KUKA KRL program: MyProgram_138().src

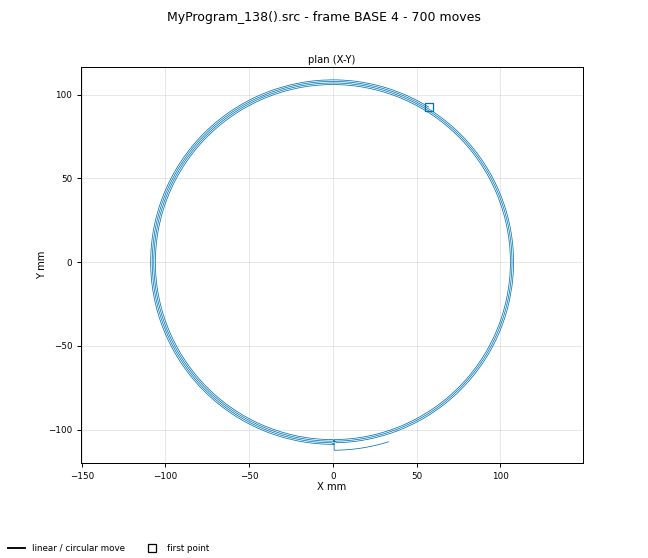
[picture p0: tool path of MyProgram_138().src in frame BASE 4, 700 of 700 moves have a stored position in this frame; points joined in program order, loops and branches not executed]
&ACCESS RVP
&REL 1
&PARAM TEMPLATE = C:\KRC\Roboter\Template\vorgabe
&PARAM EDITMASK = *
DEF MyProgram_138()
; ---- Setting reference (Base) ----
$BASE = BASE_DATA[4]

; --------------------------
; ---- Setting tool (TCP) ----
$TOOL = TOOL_DATA[3]
; --------------------------

$VEL.CP = VEL_APROX_PRINT
Startdeposition()
$VEL.CP = VEL_PRINT
LIN {X 57.2124,Y 92.5973,Z 111,A 54.04,B 24.9282,C -1.9571,E1 25.0833,E2 391.5977} C_DIS
LIN {X 54.554,Y 94.1872,Z 111,A 56.5809,B 24.9251,C -1.9983,E1 25.0769,E2 388.9668} C_DIS
LIN {X 49.9043,Y 96.7314,Z 111,A 58.528,B 24.9275,C -1.9661,E1 25.0723,E2 387.1015} C_DIS
LIN {X 44.6968,Y 99.2443,Z 111,A 61.4377,B 24.9277,C -1.9641,E1 25.065,E2 384.2041} C_DIS
LIN {X 41.4187,Y 100.6573,Z 111,A 63.4563,B 24.9271,C -1.9719,E1 25.0598,E2 382.1716} C_DIS
LIN {X 35.1577,Y 103.0113,Z 111,A 66.9301,B 24.9271,C -1.9732,E1 25.0507,E2 378.7021} C_DIS
LIN {X 31.9935,Y 104.0371,Z 111,A 68.7671,B 24.9266,C -1.9782,E1 25.0457,E2 376.8566} C_DIS
LIN {X 27.3515,Y 105.3527,Z 111,A 71.9417,B 24.9245,C -2.0064,E1 25.037,E2 373.6203} C_DIS
LIN {X 22.7022,Y 106.4523,Z 111,A 74.5175,B 24.9242,C -2.0101,E1 25.03,E2 371.0389} C_DIS
LIN {X 17.8344,Y 107.374,Z 111,A 76.2427,B 24.9269,C -1.9744,E1 25.0255,E2 369.4002} C_DIS
LIN {X 13.2214,Y 108.0405,Z 111,A 78.8231,B 24.9265,C -1.9802,E1 25.0183,E2 366.8082} C_DIS
LIN {X 10.1489,Y 108.3709,Z 111,A 80.4425,B 24.9265,C -1.9802,E1 25.0138,E2 365.1901} C_DIS
LIN {X 6.1973,Y 108.6686,Z 111,A 82.3574,B 24.927,C -1.9732,E1 25.0085,E2 363.2924} C_DIS
LIN {X 2.4816,Y 108.8177,Z 111,A 84.5086,B 24.9264,C -1.9809,E1 25.0024,E2 361.1235} C_DIS
LIN {X -0.9,Y 108.8415,Z 111,A 86.2853,B 24.9264,C -1.9804,E1 24.9975,E2 359.348} C_DIS
LIN {X -6.1677,Y 108.6702,Z 111,A 88.9687,B 24.9268,C -1.9758,E1 24.99,E2 356.675} C_DIS
LIN {X -8.9603,Y 108.4759,Z 111,A 90.5818,B 24.9264,C -1.9807,E1 24.9855,E2 355.0494} C_DIS
LIN {X -12.5967,Y 108.1136,Z 111,A 92.3889,B 24.9269,C -1.975,E1 24.9805,E2 353.2548} C_DIS
LIN {X -15.0336,Y 107.8021,Z 111,A 94.1095,B 24.9256,C -1.9914,E1 24.9757,E2 351.494} C_DIS
LIN {X -18.3991,Y 107.2796,Z 111,A 95.5312,B 24.9269,C -1.9751,E1 24.9718,E2 350.1095} C_DIS
LIN {X -25.1527,Y 105.9009,Z 111,A 99.3647,B 24.9265,C -1.9801,E1 24.9613,E2 346.2595} C_DIS
LIN {X -33.6723,Y 103.5057,Z 111,A 103.7876,B 24.9276,C -1.9656,E1 24.9496,E2 341.8638} C_DIS
LIN {X -37.933,Y 102.0233,Z 111,A 107.1546,B 24.9249,C -2.0019,E1 24.9405,E2 338.4036} C_DIS
LIN {X -43.1716,Y 99.9178,Z 111,A 109.1699,B 24.928,C -1.9597,E1 24.9355,E2 336.484} C_DIS
LIN {X -45.8586,Y 98.7129,Z 111,A 111.3295,B 24.9264,C -1.9813,E1 24.9299,E2 334.2676} C_DIS
LIN {X -49.6292,Y 96.872,Z 111,A 113.0255,B 24.9282,C -1.9575,E1 24.9258,E2 332.6237} C_DIS
LIN {X -53.729,Y 94.6613,Z 111,A 115.5042,B 24.9284,C -1.9543,E1 24.9198,E2 330.1455} C_DIS
LIN {X -56.0407,Y 93.3113,Z 111,A 117.2675,B 24.9276,C -1.9655,E1 24.9155,E2 328.3501} C_DIS
LIN {X -58.9868,Y 91.4759,Z 111,A 119.0332,B 24.928,C -1.9596,E1 24.9114,E2 326.5927} C_DIS
LIN {X -61.7031,Y 89.6661,Z 111,A 120.854,B 24.928,C -1.9602,E1 24.9072,E2 324.7644} C_DIS
LIN {X -64.732,Y 87.5059,Z 111,A 122.4158,B 24.9294,C -1.9407,E1 24.9037,E2 323.2435} C_DIS
LIN {X -66.7485,Y 85.9768,Z 111,A 124.0953,B 24.9286,C -1.9513,E1 24.9,E2 321.5326} C_DIS
LIN {X -69.373,Y 83.873,Z 111,A 126.0861,B 24.9283,C -1.9559,E1 24.8956,E2 319.5231} C_DIS
LIN {X -72.5974,Y 81.0977,Z 111,A 127.7779,B 24.9302,C -1.9296,E1 24.8922,E2 317.8873} C_DIS
LIN {X -74.913,Y 78.9651,Z 111,A 130.0033,B 24.9289,C -1.9476,E1 24.8876,E2 315.6099} C_DIS
LIN {X -77.9708,Y 75.9481,Z 111,A 132.276,B 24.9293,C -1.9425,E1 24.8832,E2 313.3397} C_DIS
LIN {X -80.856,Y 72.8675,Z 111,A 133.8967,B 24.9313,C -1.9138,E1 24.8803,E2 311.7802} C_DIS
LIN {X -83.2813,Y 70.0844,Z 111,A 136.3565,B 24.9303,C -1.9285,E1 24.8757,E2 309.2742} C_DIS
LIN {X -85.66,Y 67.1548,Z 111,A 138.0787,B 24.9314,C -1.9131,E1 24.8728,E2 307.5805} C_DIS
LIN {X -89.1664,Y 62.4237,Z 111,A 140.7257,B 24.9332,C -1.8874,E1 24.8685,E2 304.9819} C_DIS
LIN {X -92.2646,Y 57.745,Z 111,A 143.568,B 24.9341,C -1.8748,E1 24.8642,E2 302.1553} C_DIS
LIN {X -94.6562,Y 53.7379,Z 111,A 146.4084,B 24.9336,C -1.8821,E1 24.8601,E2 299.2828} C_DIS
LIN {X -96.2307,Y 50.8616,Z 111,A 147.9789,B 24.9344,C -1.8712,E1 24.8581,E2 297.73} C_DIS
LIN {X -98.007,Y 47.3488,Z 111,A 150.5224,B 24.9335,C -1.8828,E1 24.8549,E2 295.1451} C_DIS
LIN {X -99.9574,Y 43.0809,Z 111,A 152.8141,B 24.9346,C -1.8685,E1 24.8523,E2 292.875} C_DIS
LIN {X -101.0893,Y 40.3553,Z 111,A 154.9142,B 24.9334,C -1.8844,E1 24.8501,E2 290.7251} C_DIS
LIN {X -102.593,Y 36.3596,Z 111,A 156.5128,B 24.9356,C -1.8529,E1 24.8486,E2 289.1927} C_DIS
LIN {X -103.8004,Y 32.7566,Z 111,A 159.3428,B 24.9339,C -1.878,E1 24.8462,E2 286.2866} C_DIS
LIN {X -105.1746,Y 28.0297,Z 111,A 161.1618,B 24.9365,C -1.8405,E1 24.8449,E2 284.5465} C_DIS
LIN {X -105.9982,Y 24.732,Z 111,A 162.9892,B 24.9368,C -1.8362,E1 24.8437,E2 282.7186} C_DIS
LIN {X -106.7148,Y 21.4336,Z 111,A 164.5554,B 24.9377,C -1.8226,E1 24.8428,E2 281.1756} C_DIS
LIN {X -107.3259,Y 18.1224,Z 111,A 166.8034,B 24.9369,C -1.8348,E1 24.8417,E2 278.8852} C_DIS
LIN {X -107.9826,Y 13.6782,Z 111,A 168.8208,B 24.9383,C -1.8141,E1 24.8409,E2 276.9052} C_DIS
LIN {X -108.6273,Y 6.8942,Z 111,A 172.2213,B 24.9396,C -1.7953,E1 24.8401,E2 273.5289} C_DIS
LIN {X -108.8458,Y 0.346,Z 111,A 176.3293,B 24.9387,C -1.8089,E1 24.8398,E2 269.364} C_DIS
LIN {X -108.7341,Y -4.9176,Z 111,A 179.5942,B 24.938,C -1.8187,E1 24.8402,E2 266.0559} C_DIS
LIN {X -108.3957,Y -9.8796,Z 111,A -178.6874,B 24.9409,C -1.7762,E1 24.8405,E2 264.4286} C_DIS
LIN {X -108.0842,Y -12.8483,Z 111,A -176.3822,B 24.9393,C -1.7989,E1 24.8413,E2 262.0553} C_DIS
LIN {X -107.5085,Y -17.0089,Z 111,A -175.2974,B 24.9426,C -1.7494,E1 24.8417,E2 261.0822} C_DIS
LIN {X -106.7448,Y -21.2874,Z 111,A -172.4521,B 24.9417,C -1.763,E1 24.8432,E2 258.1875} C_DIS
LIN {X -106.0513,Y -24.5023,Z 111,A -170.6918,B 24.942,C -1.7588,E1 24.8442,E2 256.4271} C_DIS
LIN {X -105.1166,Y -28.2445,Z 111,A -168.6801,B 24.9425,C -1.7518,E1 24.8456,E2 254.4202} C_DIS
LIN {X -104.1481,Y -31.6353,Z 111,A -166.8566,B 24.9429,C -1.7449,E1 24.8471,E2 252.6026} C_DIS
LIN {X -103.1613,Y -34.7129,Z 111,A -165.0914,B 24.9431,C -1.7422,E1 24.8486,E2 250.8337} C_DIS
LIN {X -101.8747,Y -38.3253,Z 111,A -163.07,B 24.9435,C -1.7363,E1 24.8505,E2 248.815} C_DIS
LIN {X -99.6824,Y -43.7115,Z 111,A -159.3421,B 24.9424,C -1.753,E1 24.8547,E2 245.0267} C_DIS
LIN {X -97.851,Y -47.6734,Z 111,A -157.5507,B 24.9441,C -1.727,E1 24.8568,E2 243.2875} C_DIS
LIN {X -96.043,Y -51.2181,Z 111,A -155.4476,B 24.9445,C -1.7216,E1 24.8595,E2 241.1863} C_DIS
LIN {X -94.3257,Y -54.313,Z 111,A -153.7803,B 24.9453,C -1.709,E1 24.8617,E2 239.54} C_DIS
LIN {X -92.4096,Y -57.5128,Z 111,A -151.6872,B 24.9453,C -1.7088,E1 24.8648,E2 237.4368} C_DIS
LIN {X -90.4268,Y -60.584,Z 111,A -149.6454,B 24.9453,C -1.7083,E1 24.868,E2 235.3858} C_DIS
LIN {X -88.0816,Y -63.9457,Z 111,A -147.5847,B 24.9459,C -1.6992,E1 24.8713,E2 233.3369} C_DIS
LIN {X -85.695,Y -67.1106,Z 111,A -145.4349,B 24.9461,C -1.6965,E1 24.8749,E2 231.1831} C_DIS
LIN {X -83.4977,Y -69.8247,Z 111,A -143.7557,B 24.9467,C -1.6861,E1 24.8779,E2 229.5211} C_DIS
LIN {X -79.5983,Y -74.2398,Z 111,A -140.4764,B 24.9467,C -1.6859,E1 24.884,E2 226.2275} C_DIS
LIN {X -77.1504,Y -76.7802,Z 111,A -138.7372,B 24.9473,C -1.6773,E1 24.8874,E2 224.5013} C_DIS
LIN {X -74.6706,Y -79.1931,Z 111,A -136.8281,B 24.9473,C -1.677,E1 24.8913,E2 222.5852} C_DIS
LIN {X -71.8231,Y -81.7849,Z 111,A -134.7808,B 24.9475,C -1.6737,E1 24.8955,E2 220.5374} C_DIS
LIN {X -69.7427,Y -83.5658,Z 111,A -132.6222,B 24.9459,C -1.6994,E1 24.9003,E2 218.3096} C_DIS
LIN {X -65.9899,Y -86.5614,Z 111,A -130.9059,B 24.9482,C -1.6626,E1 24.9039,E2 216.6744} C_DIS
LIN {X -63.1094,Y -88.6818,Z 111,A -129.01,B 24.9484,C -1.6599,E1 24.9082,E2 214.7784} C_DIS
LIN {X -59.8794,Y -90.8938,Z 111,A -126.8554,B 24.9484,C -1.6603,E1 24.9132,E2 212.6157} C_DIS
LIN {X -57.6029,Y -92.3533,Z 111,A -124.5906,B 24.9464,C -1.6918,E1 24.9188,E2 210.2688} C_DIS
LIN {X -53.1291,Y -94.9975,Z 111,A -122.724,B 24.9488,C -1.653,E1 24.9231,E2 208.4889} C_DIS
LIN {X -50.1806,Y -96.5888,Z 111,A -120.7064,B 24.9483,C -1.6608,E1 24.9281,E2 206.4471} C_DIS
LIN {X -46.4955,Y -98.4164,Z 111,A -118.5097,B 24.9483,C -1.6595,E1 24.9337,E2 204.2479} C_DIS
LIN {X -42.476,Y -100.2151,Z 111,A -115.6875,B 24.9473,C -1.6775,E1 24.9411,E2 201.3763} C_DIS
LIN {X -37.9906,Y -102.0015,Z 111,A -113.8181,B 24.9491,C -1.6478,E1 24.9458,E2 199.5738} C_DIS
LIN {X -34.7676,Y -103.1428,Z 111,A -112.0211,B 24.9492,C -1.6462,E1 24.9505,E2 197.7772} C_DIS
LIN {X -31.6974,Y -104.1289,Z 111,A -110.4301,B 24.9496,C -1.6406,E1 24.9547,E2 196.1967} C_DIS
LIN {X -27.4497,Y -105.3275,Z 111,A -108.0258,B 24.9495,C -1.6424,E1 24.9612,E2 193.7843} C_DIS
LIN {X -20.9541,Y -106.8096,Z 111,A -104.6866,B 24.95,C -1.6338,E1 24.9703,E2 190.4613} C_DIS
LIN {X -17.1155,Y -107.492,Z 111,A -102.4094,B 24.9495,C -1.6424,E1 24.9766,E2 188.1616} C_DIS
LIN {X -13.3228,Y -108.0286,Z 111,A -100.3774,B 24.9495,C -1.6426,E1 24.9822,E2 186.1274} C_DIS
LIN {X -9.7573,Y -108.407,Z 111,A -98.512,B 24.9495,C -1.6416,E1 24.9874,E2 184.2635} C_DIS
LIN {X -6.19,Y -108.669,Z 111,A -96.7152,B 24.9497,C -1.6381,E1 24.9924,E2 182.4744} C_DIS
LIN {X -2.5967,Y -108.8156,Z 111,A -94.7193,B 24.9494,C -1.6426,E1 24.998,E2 180.4676} C_DIS
LIN {X 0.7454,Y -108.8411,Z 111,A -93.1023,B 24.9498,C -1.6371,E1 25.0025,E2 178.8636} C_DIS
Enddeposition()
LIN {X 0.7454,Y -108.8411,Z 111,A -93.1023,B 24.9498,C -1.6371,E1 25.0025,E2 178.8636} C_DIS
Startdeposition()
$VEL.CP = VEL_PRINT
LIN {X -0.738,Y -107.9051,Z 111,A -94.6413,B 24.9507,C -1.6223,E1 24.9981,E2 180.4376} C_DIS
LIN {X -4.3276,Y -107.8213,Z 111,A -96.6193,B 24.9509,C -1.6192,E1 24.9925,E2 182.4233} C_DIS
LIN {X -7.8193,Y -107.6253,Z 111,A -98.4701,B 24.9509,C -1.6193,E1 24.9874,E2 184.2744} C_DIS
LIN {X -11.2609,Y -107.3185,Z 111,A -100.1986,B 24.9506,C -1.6238,E1 24.9826,E2 185.9932} C_DIS
LIN {X -14.047,Y -106.9896,Z 111,A -101.7202,B 24.9506,C -1.6228,E1 24.9784,E2 187.5184} C_DIS
LIN {X -18.1316,Y -106.374,Z 111,A -103.9669,B 24.9508,C -1.6212,E1 24.9722,E2 189.7707} C_DIS
LIN {X -23.6715,Y -105.2811,Z 111,A -106.8512,B 24.9504,C -1.627,E1 24.9643,E2 192.6447} C_DIS
LIN {X -29.1742,Y -103.8893,Z 111,A -109.9817,B 24.9506,C -1.6242,E1 24.9558,E2 195.7865} C_DIS
LIN {X -32.344,Y -102.947,Z 111,A -111.6626,B 24.9503,C -1.6284,E1 24.9513,E2 197.4602} C_DIS
LIN {X -35.3965,Y -101.9376,Z 111,A -113.4529,B 24.9504,C -1.6265,E1 24.9466,E2 199.2583} C_DIS
LIN {X -38.4461,Y -100.8267,Z 111,A -115.561,B 24.9512,C -1.613,E1 24.941,E2 201.4029} C_DIS
LIN {X -41.5207,Y -99.6005,Z 111,A -117.0017,B 24.9504,C -1.6272,E1 24.9373,E2 202.8132} C_DIS
LIN {X -45.2004,Y -97.9853,Z 111,A -119.114,B 24.9502,C -1.6304,E1 24.932,E2 204.9229} C_DIS
LIN {X -48.3907,Y -96.4494,Z 111,A -120.8123,B 24.9496,C -1.6398,E1 24.9278,E2 206.6033} C_DIS
LIN {X -50.5517,Y -95.3346,Z 111,A -122.1778,B 24.9496,C -1.6386,E1 24.9244,E2 207.9754} C_DIS
LIN {X -53.5282,Y -93.6956,Z 111,A -124.5217,B 24.9508,C -1.6202,E1 24.9185,E2 210.3699} C_DIS
LIN {X -56.6609,Y -91.8366,Z 111,A -125.887,B 24.9493,C -1.645,E1 24.9154,E2 211.6805} C_DIS
LIN {X -59.0124,Y -90.3427,Z 111,A -127.9307,B 24.9505,C -1.6256,E1 24.9105,E2 213.7769} C_DIS
LIN {X -61.8911,Y -88.3951,Z 111,A -129.5546,B 24.9498,C -1.6372,E1 24.9068,E2 215.3789} C_DIS
LIN {X -65.3162,Y -85.8967,Z 111,A -132.1133,B 24.9503,C -1.6294,E1 24.9011,E2 217.9652} C_DIS
LIN {X -68.1893,Y -83.6313,Z 111,A -133.7977,B 24.9494,C -1.6429,E1 24.8975,E2 219.6239} C_DIS
LIN {X -70.9889,Y -81.2689,Z 111,A -135.4897,B 24.9486,C -1.6563,E1 24.8939,E2 221.2906} C_DIS
LIN {X -73.785,Y -78.7392,Z 111,A -137.4949,B 24.9483,C -1.6602,E1 24.8898,E2 223.2946} C_DIS
LIN {X -76.3182,Y -76.289,Z 111,A -139.5037,B 24.9484,C -1.6589,E1 24.8858,E2 225.3149} C_DIS
LIN {X -78.7402,Y -73.784,Z 111,A -141.8483,B 24.9493,C -1.6444,E1 24.8812,E2 227.7043} C_DIS
LIN {X -81.5145,Y -70.7077,Z 111,A -143.5604,B 24.9479,C -1.6677,E1 24.8782,E2 229.3686} C_DIS
LIN {X -83.3934,Y -68.4835,Z 111,A -145.1511,B 24.9478,C -1.6696,E1 24.8753,E2 230.962} C_DIS
LIN {X -85.797,Y -65.4463,Z 111,A -147.1473,B 24.9473,C -1.6769,E1 24.8719,E2 232.9504} C_DIS
LIN {X -87.9068,Y -62.5816,Z 111,A -148.9056,B 24.9467,C -1.6865,E1 24.8691,E2 234.6943} C_DIS
LIN {X -90.3725,Y -58.9672,Z 111,A -151.3572,B 24.9467,C -1.6877,E1 24.8652,E2 237.1555} C_DIS
LIN {X -92.9979,Y -54.7311,Z 111,A -153.8722,B 24.9459,C -1.6996,E1 24.8616,E2 239.655} C_DIS
LIN {X -94.4729,Y -52.1461,Z 111,A -155.6836,B 24.9461,C -1.6952,E1 24.8591,E2 241.4862} C_DIS
LIN {X -96.2263,Y -48.833,Z 111,A -157.6728,B 24.9458,C -1.7008,E1 24.8565,E2 243.4728} C_DIS
LIN {X -98.6358,Y -43.7656,Z 111,A -160.669,B 24.9453,C -1.7086,E1 24.853,E2 246.4666} C_DIS
LIN {X -100.5834,Y -39.0793,Z 111,A -163.1815,B 24.9443,C -1.7233,E1 24.8504,E2 248.9583} C_DIS
LIN {X -101.5717,Y -36.4359,Z 111,A -164.901,B 24.9446,C -1.7195,E1 24.8487,E2 250.6964} C_DIS
LIN {X -102.7174,Y -33.064,Z 111,A -166.6168,B 24.9438,C -1.7317,E1 24.8472,E2 252.393} C_DIS
LIN {X -103.7009,Y -29.839,Z 111,A -168.5725,B 24.9438,C -1.731,E1 24.8457,E2 254.3616} C_DIS
LIN {X -104.6185,Y -26.4426,Z 111,A -170.4521,B 24.9435,C -1.7363,E1 24.8444,E2 256.2395} C_DIS
LIN {X -105.5182,Y -22.5863,Z 111,A -172.3655,B 24.9426,C -1.7498,E1 24.8432,E2 258.132} C_DIS
LIN {X -106.0381,Y -20.0036,Z 111,A -174.1059,B 24.9431,C -1.7417,E1 24.8423,E2 259.9021} C_DIS
LIN {X -106.6664,Y -16.3207,Z 111,A -176.597,B 24.9439,C -1.7295,E1 24.8412,E2 262.437} C_DIS
LIN {X -107.2643,Y -11.7781,Z 111,A -178.288,B 24.9417,C -1.7642,E1 24.8407,E2 264.0554} C_DIS
LIN {X -107.75,Y -5.8312,Z 111,A 177.9183,B 24.9425,C -1.7517,E1 24.8399,E2 267.9018} C_DIS
LIN {X -107.89,Y -1.952,Z 111,A 176.4307,B 24.9407,C -1.7792,E1 24.8399,E2 269.3328} C_DIS
LIN {X -107.9017,Y 1.2877,Z 111,A 173.8525,B 24.9424,C -1.7536,E1 24.8399,E2 271.9876} C_DIS
LIN {X -107.7322,Y 6.154,Z 111,A 172.5435,B 24.9387,C -1.8084,E1 24.84,E2 273.1736} C_DIS
LIN {X -107.2342,Y 12.0474,Z 111,A 168.9032,B 24.9393,C -1.8002,E1 24.8409,E2 276.8555} C_DIS
LIN {X -106.4571,Y 17.6345,Z 111,A 165.8379,B 24.9388,C -1.8073,E1 24.8422,E2 279.922} C_DIS
LIN {X -105.8443,Y 21.0099,Z 111,A 164.0175,B 24.9384,C -1.8132,E1 24.8431,E2 281.7393} C_DIS
LIN {X -105.1387,Y 24.2879,Z 111,A 162.2901,B 24.9379,C -1.8208,E1 24.8442,E2 283.4585} C_DIS
LIN {X -104.3811,Y 27.3664,Z 111,A 160.6393,B 24.9374,C -1.8274,E1 24.8453,E2 285.1033} C_DIS
LIN {X -102.9089,Y 32.4669,Z 111,A 157.825,B 24.9368,C -1.8364,E1 24.8475,E2 287.9123} C_DIS
LIN {X -102.0759,Y 34.9982,Z 111,A 155.8643,B 24.9378,C -1.8209,E1 24.8493,E2 289.9212} C_DIS
LIN {X -100.9575,Y 38.1006,Z 111,A 154.5126,B 24.9365,C -1.8409,E1 24.8506,E2 291.2327} C_DIS
LIN {X -99.5516,Y 41.6369,Z 111,A 152.4306,B 24.9362,C -1.8449,E1 24.8528,E2 293.3169} C_DIS
LIN {X -98.0253,Y 45.1144,Z 111,A 150.432,B 24.9357,C -1.8517,E1 24.8551,E2 295.3103} C_DIS
LIN {X -95.5364,Y 50.1685,Z 111,A 147.6057,B 24.9347,C -1.8666,E1 24.8586,E2 298.1161} C_DIS
LIN {X -94.2246,Y 52.5907,Z 111,A 145.5303,B 24.936,C -1.8485,E1 24.8614,E2 300.2458} C_DIS
LIN {X -92.4493,Y 55.6543,Z 111,A 144.2671,B 24.934,C -1.8765,E1 24.8632,E2 301.4486} C_DIS
LIN {X -89.2122,Y 60.7067,Z 111,A 140.9249,B 24.9338,C -1.8797,E1 24.8683,E2 304.7999} C_DIS
LIN {X -85.9122,Y 65.2936,Z 111,A 137.8999,B 24.9332,C -1.887,E1 24.8732,E2 307.8223} C_DIS
LIN {X -83.5498,Y 68.2912,Z 111,A 135.9664,B 24.9326,C -1.8958,E1 24.8766,E2 309.7439} C_DIS
LIN {X -81.9069,Y 70.2527,Z 111,A 134.3441,B 24.9331,C -1.8896,E1 24.8795,E2 311.3885} C_DIS
LIN {X -79.3749,Y 73.1007,Z 111,A 132.1113,B 24.9333,C -1.8869,E1 24.8838,E2 313.6374} C_DIS
LIN {X -75.2518,Y 77.3401,Z 111,A 129.2233,B 24.932,C -1.9039,E1 24.8894,E2 316.4973} C_DIS
LIN {X -72.8042,Y 79.647,Z 111,A 127.2477,B 24.9322,C -1.9011,E1 24.8935,E2 318.4877} C_DIS
LIN {X -68.7496,Y 83.1723,Z 111,A 124.4574,B 24.9316,C -1.9098,E1 24.8994,E2 321.268} C_DIS
LIN {X -66.5195,Y 84.9674,Z 111,A 122.9827,B 24.9313,C -1.9148,E1 24.9026,E2 322.7363} C_DIS
LIN {X -63.6498,Y 87.1366,Z 111,A 120.3678,B 24.9329,C -1.8925,E1 24.9087,E2 325.4135} C_DIS
LIN {X -59.63,Y 89.9355,Z 111,A 118.7898,B 24.9297,C -1.9359,E1 24.9121,E2 326.8934} C_DIS
LIN {X -55.5862,Y 92.4906,Z 111,A 116.0946,B 24.9298,C -1.9348,E1 24.9185,E2 329.5999} C_DIS
LIN {X -53.447,Y 93.7422,Z 111,A 114.6018,B 24.9301,C -1.9304,E1 24.9221,E2 331.1075} C_DIS
LIN {X -48.8756,Y 96.2045,Z 111,A 111.429,B 24.9309,C -1.9193,E1 24.93,E2 334.3153} C_DIS
LIN {X -45.6455,Y 97.7781,Z 111,A 110.3349,B 24.9285,C -1.9533,E1 24.9326,E2 335.3315} C_DIS
LIN {X -38.3358,Y 100.8684,Z 111,A 105.8393,B 24.9288,C -1.9485,E1 24.9443,E2 339.8488} C_DIS
LIN {X -35.4539,Y 101.9174,Z 111,A 104.1595,B 24.9288,C -1.9485,E1 24.9487,E2 341.5317} C_DIS
LIN {X -30.921,Y 103.3828,Z 111,A 101.238,B 24.9297,C -1.9364,E1 24.9565,E2 344.4873} C_DIS
LIN {X -27.1414,Y 104.4389,Z 111,A 99.472,B 24.9287,C -1.9508,E1 24.9612,E2 346.2218} C_DIS
LIN {X -23.6603,Y 105.2837,Z 111,A 97.4588,B 24.9288,C -1.9482,E1 24.9667,E2 348.2438} C_DIS
LIN {X -19.8949,Y 106.059,Z 111,A 95.7104,B 24.9279,C -1.9613,E1 24.9714,E2 349.9631} C_DIS
LIN {X -14.7588,Y 106.8944,Z 111,A 92.8831,B 24.9279,C -1.9606,E1 24.9793,E2 352.7943} C_DIS
LIN {X -11.7408,Y 107.2682,Z 111,A 91.0802,B 24.9284,C -1.9542,E1 24.9843,E2 354.6138} C_DIS
LIN {X -8.2886,Y 107.5893,Z 111,A 89.3773,B 24.9279,C -1.9605,E1 24.989,E2 356.3025} C_DIS
LIN {X -4.4317,Y 107.8168,Z 111,A 87.1143,B 24.9285,C -1.9529,E1 24.9954,E2 358.5842} C_DIS
LIN {X -0.4353,Y 107.907,Z 111,A 85.1947,B 24.9279,C -1.9614,E1 25.0007,E2 360.4836} C_DIS
LIN {X 2.8838,Y 107.8693,Z 111,A 83.4912,B 24.9277,C -1.964,E1 25.0054,E2 362.1807} C_DIS
LIN {X 5.0706,Y 107.7893,Z 111,A 82.2144,B 24.928,C -1.9595,E1 25.009,E2 363.4679} C_DIS
LIN {X 8.5205,Y 107.5707,Z 111,A 80.419,B 24.9279,C -1.961,E1 25.014,E2 365.2587} C_DIS
LIN {X 11.9578,Y 107.2447,Z 111,A 78.184,B 24.9291,C -1.9447,E1 25.0203,E2 367.5308} C_DIS
LIN {X 16.6099,Y 106.6217,Z 111,A 75.8193,B 24.9288,C -1.9492,E1 25.0268,E2 369.8829} C_DIS
LIN {X 21.239,Y 105.7978,Z 111,A 73.4981,B 24.9283,C -1.9552,E1 25.0331,E2 372.1873} C_DIS
LIN {X 26.4088,Y 104.6272,Z 111,A 70.6942,B 24.9284,C -1.954,E1 25.0407,E2 374.9899} C_DIS
LIN {X 29.5337,Y 103.7875,Z 111,A 69.0654,B 24.9282,C -1.9565,E1 25.0451,E2 376.6102} C_DIS
LIN {X 32.6151,Y 102.8626,Z 111,A 67.2668,B 24.9286,C -1.9515,E1 25.0499,E2 378.4174} C_DIS
LIN {X 35.6864,Y 101.8359,Z 111,A 65.2529,B 24.9296,C -1.9381,E1 25.0553,E2 380.4591} C_DIS
LIN {X 38.7765,Y 100.7015,Z 111,A 63.9576,B 24.9284,C -1.9548,E1 25.0586,E2 381.712} C_DIS
LIN {X 42.2315,Y 99.301,Z 111,A 61.9507,B 24.9286,C -1.9516,E1 25.0638,E2 383.7218} C_DIS
LIN {X 46.2111,Y 97.5133,Z 111,A 59.738,B 24.9285,C -1.9531,E1 25.0694,E2 385.9253} C_DIS
LIN {X 48.5885,Y 96.3512,Z 111,A 58.086,B 24.9294,C -1.9412,E1 25.0735,E2 387.6012} C_DIS
LIN {X 53.6524,Y 93.6242,Z 111,A 55.1647,B 24.9293,C -1.9425,E1 25.0807,E2 390.511} C_DIS
LIN {X 56.3715,Y 92.0134,Z 111,A 53.3292,B 24.9299,C -1.9334,E1 25.0851,E2 392.3622} C_DIS
LIN {X 59.719,Y 89.8769,Z 111,A 51.2986,B 24.9299,C -1.9333,E1 25.0898,E2 394.3865} C_DIS
LIN {X 62.5438,Y 87.9338,Z 111,A 49.5654,B 24.9299,C -1.9338,E1 25.0938,E2 396.1123} C_DIS
LIN {X 65.2492,Y 85.9471,Z 111,A 47.6885,B 24.9304,C -1.9267,E1 25.098,E2 397.9994} C_DIS
LIN {X 69.1918,Y 82.8048,Z 111,A 45.2182,B 24.9301,C -1.9303,E1 25.1033,E2 400.4517} C_DIS
LIN {X 71.2958,Y 81.0009,Z 111,A 43.6626,B 24.9306,C -1.9239,E1 25.1066,E2 402.0165} C_DIS
LIN {X 73.9316,Y 78.6014,Z 111,A 41.802,B 24.9308,C -1.9214,E1 25.1104,E2 403.8754} C_DIS
LIN {X 76.3037,Y 76.3037,Z 111,A 39.9056,B 24.9315,C -1.9116,E1 25.1142,E2 405.787} C_DIS
LIN {X 78.694,Y 73.8332,Z 111,A 38.1583,B 24.9315,C -1.9109,E1 25.1176,E2 407.5284} C_DIS
LIN {X 81.3051,Y 70.9475,Z 111,A 36.1391,B 24.9317,C -1.9081,E1 25.1213,E2 409.545} C_DIS
LIN {X 83.7948,Y 67.989,Z 111,A 34.1002,B 24.932,C -1.9039,E1 25.125,E2 411.5846} C_DIS
LIN {X 86.0865,Y 65.0636,Z 111,A 32.1213,B 24.9324,C -1.8988,E1 25.1283,E2 413.566} C_DIS
LIN {X 88.6392,Y 61.5399,Z 111,A 29.886,B 24.9326,C -1.8962,E1 25.132,E2 415.7966} C_DIS
LIN {X 89.9593,Y 59.5939,Z 111,A 28.6161,B 24.9329,C -1.8921,E1 25.1339,E2 417.07} C_DIS
LIN {X 91.5625,Y 57.0998,Z 111,A 27.0118,B 24.9333,C -1.8866,E1 25.1363,E2 418.679} C_DIS
LIN {X 94.2304,Y 52.5803,Z 111,A 24.3994,B 24.9333,C -1.8866,E1 25.14,E2 421.2781} C_DIS
LIN {X 95.6737,Y 49.9077,Z 111,A 22.4295,B 24.9347,C -1.8668,E1 25.1426,E2 423.2843} C_DIS
LIN {X 98.0946,Y 44.9656,Z 111,A 19.7273,B 24.9346,C -1.8679,E1 25.1458,E2 425.9693} C_DIS
LIN {X 99.4483,Y 41.8818,Z 111,A 18.0013,B 24.9348,C -1.8655,E1 25.1477,E2 427.6917} C_DIS
LIN {X 100.7789,Y 38.5723,Z 111,A 15.9223,B 24.9357,C -1.8519,E1 25.1499,E2 429.7911} C_DIS
LIN {X 102.3459,Y 34.1973,Z 111,A 13.6726,B 24.9356,C -1.8539,E1 25.1519,E2 432.0234} C_DIS
LIN {X 103.5566,Y 30.3352,Z 111,A 10.857,B 24.938,C -1.8187,E1 25.1542,E2 434.9061} C_DIS
LIN {X 104.7105,Y 26.0776,Z 111,A 9.3373,B 24.9361,C -1.8469,E1 25.1553,E2 436.3504} C_DIS
LIN {X 105.6823,Y 21.802,Z 111,A 6.4794,B 24.9381,C -1.8167,E1 25.157,E2 439.2629} C_DIS
LIN {X 106.3218,Y 18.4435,Z 111,A 4.9475,B 24.9377,C -1.8232,E1 25.1577,E2 440.7706} C_DIS
LIN {X 106.9433,Y 14.4042,Z 111,A 3.0533,B 24.9373,C -1.8283,E1 25.1585,E2 442.6415} C_DIS
LIN {X 107.4354,Y 10.086,Z 111,A 0.6302,B 24.9382,C -1.8159,E1 25.1592,E2 445.0795} C_DIS
LIN {X 107.6816,Y 6.987,Z 111,A -1.1243,B 24.9389,C -1.8061,E1 25.1595,E2 446.8468} C_DIS
LIN {X 107.8569,Y 3.3087,Z 111,A -2.9103,B 24.9388,C -1.8072,E1 25.1597,E2 448.6196} C_DIS
LIN {X 107.9106,Y 0.0081,Z 111,A -4.8343,B 24.9397,C -1.794,E1 25.1597,E2 450.5633} C_DIS
LIN {X 107.842,Y -3.7943,Z 111,A -6.7379,B 24.9397,C -1.7925,E1 25.1597,E2 452.4591} C_DIS
LIN {X 107.6659,Y -7.2186,Z 111,A -8.5067,B 24.94,C -1.7888,E1 25.1593,E2 454.226} C_DIS
LIN {X 107.3472,Y -10.9862,Z 111,A -10.523,B 24.9405,C -1.7819,E1 25.1588,E2 456.2466} C_DIS
LIN {X 106.9455,Y -14.3875,Z 111,A -12.4959,B 24.9413,C -1.7693,E1 25.1581,E2 458.2377} C_DIS
LIN {X 105.4909,Y -22.7113,Z 111,A -16.5089,B 24.9409,C -1.7755,E1 25.1562,E2 462.2126} C_DIS
LIN {X 104.4457,Y -27.115,Z 111,A -19.0926,B 24.942,C -1.7599,E1 25.1544,E2 464.8182} C_DIS
LIN {X 103.8442,Y -29.3333,Z 111,A -20.3649,B 24.9424,C -1.7537,E1 25.1535,E2 466.0976} C_DIS
LIN {X 102.9047,Y -32.4804,Z 111,A -21.9992,B 24.9424,C -1.753,E1 25.1521,E2 467.7244} C_DIS
LIN {X 101.6954,Y -36.0867,Z 111,A -24.6286,B 24.9445,C -1.7202,E1 25.1497,E2 470.4164} C_DIS
LIN {X 100.3576,Y -39.6542,Z 111,A -26.1254,B 24.9435,C -1.7367,E1 25.1482,E2 471.8659} C_DIS
LIN {X 99.1494,Y -42.5887,Z 111,A -28.2204,B 24.945,C -1.7137,E1 25.1459,E2 474.0036} C_DIS
LIN {X 97.7747,Y -45.6529,Z 111,A -29.5044,B 24.9439,C -1.73,E1 25.1444,E2 475.2423} C_DIS
LIN {X 96.3857,Y -48.5209,Z 111,A -31.7511,B 24.9458,C -1.7008,E1 25.1416,E2 477.5458} C_DIS
LIN {X 94.6609,Y -51.8028,Z 111,A -33.1101,B 24.9445,C -1.7214,E1 25.1398,E2 478.8491} C_DIS
LIN {X 93.0872,Y -54.58,Z 111,A -34.8665,B 24.945,C -1.7138,E1 25.1374,E2 480.6144} C_DIS
LIN {X 91.0387,Y -57.9327,Z 111,A -37.6636,B 24.9473,C -1.6771,E1 25.1331,E2 483.4838} C_DIS
LIN {X 88.5039,Y -61.7345,Z 111,A -39.3636,B 24.9457,C -1.7016,E1 25.1305,E2 485.1177} C_DIS
LIN {X 84.8324,Y -66.6903,Z 111,A -42.3568,B 24.9455,C -1.7048,E1 25.1256,E2 488.089} C_DIS
LIN {X 80.6833,Y -71.6551,Z 111,A -46.0222,B 24.9467,C -1.6858,E1 25.1189,E2 491.7826} C_DIS
LIN {X 76.0688,Y -76.5357,Z 111,A -50.3761,B 24.9494,C -1.6433,E1 25.1102,E2 496.218} C_DIS
LIN {X 72.4483,Y -79.9732,Z 111,A -52.3282,B 24.9479,C -1.6667,E1 25.1064,E2 498.1069} C_DIS
LIN {X 67.3844,Y -84.2838,Z 111,A -55.9246,B 24.9486,C -1.656,E1 25.0986,E2 501.7149} C_DIS
LIN {X 64.2159,Y -86.7221,Z 111,A -57.7313,B 24.9481,C -1.6649,E1 25.0947,E2 503.4939} C_DIS
LIN {X 58.5115,Y -90.6671,Z 111,A -61.6113,B 24.949,C -1.6491,E1 25.0857,E2 507.3982} C_DIS
LIN {X 55.5622,Y -92.5052,Z 111,A -63.4501,B 24.9492,C -1.6459,E1 25.0813,E2 509.2389} C_DIS
LIN {X 52.5474,Y -94.2488,Z 111,A -65.8567,B 24.9509,C -1.6192,E1 25.0753,E2 511.7015} C_DIS
LIN {X 48.6146,Y -96.3378,Z 111,A -67.7018,B 24.9498,C -1.6369,E1 25.0708,E2 513.4995} C_DIS
LIN {X 42.3827,Y -99.2372,Z 111,A -71.0416,B 24.9493,C -1.6443,E1 25.0624,E2 516.8135} C_DIS
LIN {X 38.0322,Y -100.9834,Z 111,A -73.6631,B 24.9499,C -1.6352,E1 25.0555,E2 519.4506} C_DIS
LIN {X 34.7539,Y -102.1583,Z 111,A -75.5159,B 24.95,C -1.6327,E1 25.0506,E2 521.3058} C_DIS
LIN {X 31.6978,Y -103.1474,Z 111,A -77.5269,B 24.9509,C -1.618,E1 25.0452,E2 523.3479} C_DIS
LIN {X 24.2476,Y -105.1481,Z 111,A -81.3049,B 24.9504,C -1.6269,E1 25.0351,E2 527.0989} C_DIS
LIN {X 21.4218,Y -105.7603,Z 111,A -82.9754,B 24.9508,C -1.62,E1 25.0304,E2 528.7839} C_DIS
LIN {X 15.8967,Y -106.732,Z 111,A -85.7213,B 24.9504,C -1.6272,E1 25.0229,E2 531.5097} C_DIS
LIN {X 13.2093,Y -107.0981,Z 111,A -87.3335,B 24.9509,C -1.6192,E1 25.0184,E2 533.1395} C_DIS
LIN {X 9.947,Y -107.4482,Z 111,A -88.9821,B 24.9507,C -1.6221,E1 25.0139,E2 534.7802} C_DIS
LIN {X 6.2467,Y -107.7271,Z 111,A -91.015,B 24.9509,C -1.6187,E1 25.0082,E2 536.8204} C_DIS
LIN {X 2.5986,Y -107.8781,Z 111,A -92.9933,B 24.951,C -1.6164,E1 25.0026,E2 538.8037} C_DIS
LIN {X 2.5986,Y -107.8781,Z 111,A -92.9933,B 24.951,C -1.6164,E1 25.0026,E2 538.8037} C_DIS
Enddeposition()
LIN {X 0.7392,Y -106.965,Z 111,A -93.8206,B 24.9496,C -1.6392,E1 25.0005,E2 539.5768} C_DIS
Startdeposition()
$VEL.CP = VEL_PRINT
LIN {X 2.536,Y -106.9417,Z 111,A -92.2411,B 24.9481,C -1.6644,E1 25.0051,E2 537.9377} C_DIS
LIN {X 5.275,Y -106.842,Z 111,A -90.5193,B 24.9474,C -1.6754,E1 25.0099,E2 536.1905} C_DIS
LIN {X 9.3438,Y -106.5626,Z 111,A -88.4308,B 24.9476,C -1.6725,E1 25.0157,E2 534.1099} C_DIS
LIN {X 12.9354,Y -106.1865,Z 111,A -86.6457,B 24.9479,C -1.6675,E1 25.0206,E2 532.3379} C_DIS
LIN {X 16.3048,Y -105.7204,Z 111,A -84.0145,B 24.9457,C -1.7025,E1 25.0281,E2 529.6262} C_DIS
LIN {X 20.9634,Y -104.8976,Z 111,A -82.3489,B 24.9478,C -1.6684,E1 25.0325,E2 528.0435} C_DIS
LIN {X 23.9158,Y -104.2627,Z 111,A -79.5353,B 24.9445,C -1.7201,E1 25.0405,E2 525.1112} C_DIS
LIN {X 29.8014,Y -102.7364,Z 111,A -77.3853,B 24.9473,C -1.677,E1 25.046,E2 523.0669} C_DIS
LIN {X 32.3942,Y -101.9489,Z 111,A -75.7962,B 24.9468,C -1.6845,E1 25.0502,E2 521.463} C_DIS
LIN {X 36.0655,Y -100.7091,Z 111,A -73.9344,B 24.9472,C -1.6781,E1 25.0551,E2 519.6199} C_DIS
LIN {X 38.1305,Y -99.9439,Z 111,A -72.589,B 24.9467,C -1.6867,E1 25.0586,E2 518.257} C_DIS
LIN {X 41.3479,Y -98.6562,Z 111,A -70.5732,B 24.9461,C -1.6962,E1 25.0639,E2 516.2235} C_DIS
LIN {X 47.8215,Y -95.6863,Z 111,A -67.2559,B 24.947,C -1.6811,E1 25.0722,E2 512.9503} C_DIS
LIN {X 51.8391,Y -93.5707,Z 111,A -64.812,B 24.9467,C -1.6858,E1 25.0782,E2 510.5023} C_DIS
LIN {X 55.4481,Y -91.4777,Z 111,A -62.3238,B 24.9458,C -1.7007,E1 25.0843,E2 507.9865} C_DIS
LIN {X 58.247,Y -89.7231,Z 111,A -60.426,B 24.9452,C -1.7096,E1 25.0888,E2 506.0738} C_DIS
LIN {X 60.6308,Y -88.1296,Z 111,A -58.9709,B 24.9452,C -1.7093,E1 25.0921,E2 504.6245} C_DIS
LIN {X 63.5378,Y -86.0568,Z 111,A -57.1351,B 24.9452,C -1.71,E1 25.0962,E2 502.7934} C_DIS
LIN {X 66.2856,Y -83.9575,Z 111,A -55.1578,B 24.9446,C -1.7194,E1 25.1006,E2 500.8012} C_DIS
LIN {X 71.1383,Y -79.8878,Z 111,A -51.9962,B 24.9447,C -1.7172,E1 25.1073,E2 497.6571} C_DIS
LIN {X 75.5605,Y -75.7203,Z 111,A -48.8941,B 24.9447,C -1.7183,E1 25.1136,E2 494.5652} C_DIS
LIN {X 79.4119,Y -71.67,Z 111,A -45.9203,B 24.9442,C -1.725,E1 25.1193,E2 491.5886} C_DIS
LIN {X 84.2835,Y -65.8726,Z 111,A -41.4609,B 24.9424,C -1.7531,E1 25.1273,E2 487.0833} C_DIS
LIN {X 87.041,Y -62.1812,Z 111,A -39.1987,B 24.9425,C -1.751,E1 25.131,E2 484.8371} C_DIS
LIN {X 89.0917,Y -59.207,Z 111,A -37.1903,B 24.942,C -1.7596,E1 25.1341,E2 482.8183} C_DIS
LIN {X 91.0543,Y -56.1441,Z 111,A -35.2572,B 24.9416,C -1.7645,E1 25.137,E2 480.8835} C_DIS
LIN {X 93.0574,Y -52.7575,Z 111,A -33.1622,B 24.9413,C -1.7701,E1 25.1399,E2 478.786} C_DIS
LIN {X 94.8672,Y -49.4275,Z 111,A -31.4007,B 24.9417,C -1.7644,E1 25.1422,E2 477.0473} C_DIS
LIN {X 96.0232,Y -47.1419,Z 111,A -29.9626,B 24.9412,C -1.7714,E1 25.144,E2 475.6003} C_DIS
LIN {X 98.134,Y -42.5723,Z 111,A -27.3023,B 24.9407,C -1.7781,E1 25.1471,E2 472.9388} C_DIS
LIN {X 100.0201,Y -37.9291,Z 111,A -24.1465,B 24.9388,C -1.8071,E1 25.1503,E2 469.732} C_DIS
LIN {X 101.1909,Y -34.6891,Z 111,A -22.7653,B 24.9398,C -1.7924,E1 25.1516,E2 468.3932} C_DIS
LIN {X 102.0227,Y -32.16,Z 111,A -21.201,B 24.9391,C -1.803,E1 25.1529,E2 466.8128} C_DIS
LIN {X 103.1485,Y -28.3415,Z 111,A -19.0962,B 24.9387,C -1.8086,E1 25.1545,E2 464.7069} C_DIS
LIN {X 104.1716,Y -24.31,Z 111,A -17.119,B 24.939,C -1.8047,E1 25.1558,E2 462.7502} C_DIS
LIN {X 104.8257,Y -21.3135,Z 111,A -15.378,B 24.9383,C -1.8143,E1 25.1568,E2 460.9967} C_DIS
LIN {X 105.4778,Y -17.8076,Z 111,A -12.8892,B 24.9361,C -1.846,E1 25.158,E2 458.4478} C_DIS
LIN {X 106.0664,Y -13.8775,Z 111,A -11.6753,B 24.9384,C -1.8127,E1 25.1585,E2 457.3197} C_DIS
LIN {X 106.3772,Y -11.249,Z 111,A -9.9457,B 24.9372,C -1.8309,E1 25.159,E2 455.5573} C_DIS
LIN {X 106.6601,Y -8.1486,Z 111,A -8.1919,B 24.9365,C -1.8401,E1 25.1594,E2 453.7922} C_DIS
LIN {X 106.8721,Y -4.583,Z 111,A -6.3923,B 24.9365,C -1.8413,E1 25.1597,E2 452.0004} C_DIS
LIN {X 106.9545,Y -1.8447,Z 111,A -4.9784,B 24.9363,C -1.8437,E1 25.1597,E2 450.5892} C_DIS
LIN {X 106.959,Y 1.6008,Z 111,A -3.0497,B 24.9356,C -1.8534,E1 25.1597,E2 448.6493} C_DIS
LIN {X 106.8396,Y 5.3193,Z 111,A -1.2229,B 24.9356,C -1.8525,E1 25.1595,E2 446.8354} C_DIS
LIN {X 106.6732,Y 7.985,Z 111,A 0.3922,B 24.9348,C -1.8652,E1 25.1592,E2 445.1999} C_DIS
LIN {X 106.3456,Y 11.5512,Z 111,A 2.3194,B 24.9343,C -1.8718,E1 25.1587,E2 443.2686} C_DIS
LIN {X 105.4364,Y 18.0551,Z 111,A 6.5316,B 24.9314,C -1.9135,E1 25.1568,E2 438.9828} C_DIS
LIN {X 104.4777,Y 22.9582,Z 111,A 8.3243,B 24.9335,C -1.883,E1 25.1558,E2 437.2723} C_DIS
LIN {X 103.7188,Y 26.1777,Z 111,A 10.2729,B 24.9326,C -1.8962,E1 25.1545,E2 435.304} C_DIS
LIN {X 102.5136,Y 30.5553,Z 111,A 12.5331,B 24.9326,C -1.8962,E1 25.1528,E2 433.0567} C_DIS
LIN {X 101.5335,Y 33.673,Z 111,A 14.1443,B 24.9326,C -1.8954,E1 25.1514,E2 431.4566} C_DIS
LIN {X 100.5475,Y 36.5086,Z 111,A 15.8714,B 24.9319,C -1.9054,E1 25.1498,E2 429.7156} C_DIS
LIN {X 99.5254,Y 39.209,Z 111,A 17.3878,B 24.9317,C -1.9086,E1 25.1483,E2 428.1999} C_DIS
LIN {X 98.1456,Y 42.5457,Z 111,A 19.4011,B 24.9311,C -1.9177,E1 25.1461,E2 426.1763} C_DIS
LIN {X 96.6926,Y 45.7547,Z 111,A 21.6221,B 24.9296,C -1.9376,E1 25.1434,E2 423.9204} C_DIS
LIN {X 95.2702,Y 48.6439,Z 111,A 22.7259,B 24.9312,C -1.9155,E1 25.1421,E2 422.8746} C_DIS
LIN {X 93.9953,Y 51.064,Z 111,A 24.379,B 24.9303,C -1.9276,E1 25.1399,E2 421.2015} C_DIS
LIN {X 92.6152,Y 53.5271,Z 111,A 26.0067,B 24.9297,C -1.9367,E1 25.1376,E2 419.5608} C_DIS
LIN {X 90.6818,Y 56.7404,Z 111,A 27.864,B 24.9297,C -1.9355,E1 25.1349,E2 417.7158} C_DIS
LIN {X 88.5703,Y 59.9829,Z 111,A 30.4117,B 24.9279,C -1.9614,E1 25.1309,E2 415.1198} C_DIS
LIN {X 86.5144,Y 62.9129,Z 111,A 31.6261,B 24.9297,C -1.936,E1 25.129,E2 413.9711} C_DIS
LIN {X 84.2916,Y 65.8629,Z 111,A 33.9557,B 24.9283,C -1.9558,E1 25.125,E2 411.6057} C_DIS
LIN {X 81.9306,Y 68.7773,Z 111,A 35.9314,B 24.928,C -1.9591,E1 25.1215,E2 409.6313} C_DIS
LIN {X 79.5843,Y 71.4774,Z 111,A 37.7794,B 24.928,C -1.9606,E1 25.1181,E2 407.788} C_DIS
LIN {X 77.0337,Y 74.2189,Z 111,A 39.7577,B 24.9277,C -1.9639,E1 25.1143,E2 405.8106} C_DIS
LIN {X 74.3171,Y 76.9391,Z 111,A 41.7668,B 24.9275,C -1.9662,E1 25.1103,E2 403.8046} C_DIS
LIN {X 71.8296,Y 79.269,Z 111,A 43.722,B 24.9268,C -1.9754,E1 25.1062,E2 401.8356} C_DIS
LIN {X 69.0404,Y 81.7083,Z 111,A 45.7613,B 24.9264,C -1.9816,E1 25.1019,E2 399.7896} C_DIS
LIN {X 65.7144,Y 84.407,Z 111,A 47.9322,B 24.9264,C -1.9806,E1 25.0972,E2 397.6291} C_DIS
LIN {X 62.7083,Y 86.6641,Z 111,A 49.7736,B 24.9267,C -1.9769,E1 25.0931,E2 395.803} C_DIS
LIN {X 60.1234,Y 88.4752,Z 111,A 51.5135,B 24.9264,C -1.9819,E1 25.0891,E2 394.0574} C_DIS
LIN {X 56.3118,Y 90.9495,Z 111,A 53.7914,B 24.9266,C -1.9792,E1 25.0837,E2 391.7931} C_DIS
LIN {X 54.2344,Y 92.2026,Z 111,A 55.3787,B 24.9255,C -1.9931,E1 25.0799,E2 390.1778} C_DIS
LIN {X 50.715,Y 94.1846,Z 111,A 57.4294,B 24.9256,C -1.9914,E1 25.0749,E2 388.1371} C_DIS
LIN {X 47.5847,Y 95.8037,Z 111,A 59.3586,B 24.9253,C -1.9956,E1 25.07,E2 386.2034} C_DIS
LIN {X 44.3045,Y 97.3648,Z 111,A 61.2712,B 24.9253,C -1.9965,E1 25.0652,E2 384.2935} C_DIS
LIN {X 39.7184,Y 99.3253,Z 111,A 64.0354,B 24.9248,C -2.0031,E1 25.0581,E2 381.52} C_DIS
LIN {X 36.2183,Y 100.6533,Z 111,A 65.7842,B 24.9254,C -1.9945,E1 25.0535,E2 379.7953} C_DIS
LIN {X 33.5309,Y 101.5811,Z 111,A 67.3401,B 24.9252,C -1.9971,E1 25.0494,E2 378.2362} C_DIS
LIN {X 30.508,Y 102.5276,Z 111,A 69.1935,B 24.9246,C -2.0048,E1 25.0444,E2 376.3679} C_DIS
LIN {X 27.3512,Y 103.416,Z 111,A 70.9955,B 24.9244,C -2.0078,E1 25.0396,E2 374.5616} C_DIS
LIN {X 23.8937,Y 104.2678,Z 111,A 72.7457,B 24.9248,C -2.0025,E1 25.0348,E2 372.8265} C_DIS
LIN {X 20.6577,Y 104.9576,Z 111,A 74.5928,B 24.9245,C -2.0063,E1 25.0298,E2 370.9726} C_DIS
LIN {X 16.3715,Y 105.7101,Z 111,A 76.6776,B 24.9252,C -1.9972,E1 25.0241,E2 368.9116} C_DIS
LIN {X 10.9704,Y 106.4064,Z 111,A 79.836,B 24.9244,C -2.0075,E1 25.0153,E2 365.7313} C_DIS
LIN {X 7.383,Y 106.7153,Z 111,A 81.7622,B 24.9244,C -2.0075,E1 25.0099,E2 363.806} C_DIS
LIN {X 3.5742,Y 106.911,Z 111,A 84.1041,B 24.9235,C -2.0193,E1 25.0033,E2 361.4367} C_DIS
LIN {X -0.7735,Y 106.9676,Z 111,A 86.1283,B 24.9245,C -2.0067,E1 24.9977,E2 359.4425} C_DIS
LIN {X -7.1057,Y 106.7341,Z 111,A 89.479,B 24.9247,C -2.0038,E1 24.9884,E2 356.0979} C_DIS
LIN {X -10.7634,Y 106.4281,Z 111,A 91.5106,B 24.9246,C -2.0054,E1 24.9828,E2 354.0615} C_DIS
LIN {X -14.2233,Y 106.0216,Z 111,A 93.8905,B 24.9231,C -2.0246,E1 24.976,E2 351.6343} C_DIS
LIN {X -18.0681,Y 105.4342,Z 111,A 95.3328,B 24.9252,C -1.9978,E1 24.9722,E2 350.2542} C_DIS
LIN {X -20.5469,Y 104.9789,Z 111,A 96.7449,B 24.9251,C -1.9992,E1 24.9683,E2 348.8373} C_DIS
LIN {X -24.0146,Y 104.2399,Z 111,A 98.667,B 24.9251,C -1.9984,E1 24.9631,E2 346.9147} C_DIS
LIN {X -27.2852,Y 103.4338,Z 111,A 100.5449,B 24.9251,C -1.9994,E1 24.958,E2 345.0316} C_DIS
LIN {X -30.4295,Y 102.5509,Z 111,A 102.5975,B 24.9243,C -2.0094,E1 24.9524,E2 342.9521} C_DIS
LIN {X -33.4882,Y 101.5949,Z 111,A 103.8473,B 24.9258,C -1.9892,E1 24.9492,E2 341.7479} C_DIS
LIN {X -37.0122,Y 100.3638,Z 111,A 106.0538,B 24.9254,C -1.9947,E1 24.9434,E2 339.5241} C_DIS
LIN {X -41.4161,Y 98.6274,Z 111,A 108.1863,B 24.9268,C -1.9756,E1 24.938,E2 337.4321} C_DIS
LIN {X -43.9715,Y 97.5149,Z 111,A 110.0117,B 24.926,C -1.9862,E1 24.9332,E2 335.5773} C_DIS
LIN {X -46.9293,Y 96.1286,Z 111,A 111.8447,B 24.926,C -1.9866,E1 24.9286,E2 333.7386} C_DIS
LIN {X -51.8728,Y 93.5519,Z 111,A 114.7734,B 24.9265,C -1.9793,E1 24.9214,E2 330.8189} C_DIS
LIN {X -54.8568,Y 91.8348,Z 111,A 116.9756,B 24.9258,C -1.9896,E1 24.916,E2 328.5855} C_DIS
LIN {X -59.12,Y 89.149,Z 111,A 119.277,B 24.9273,C -1.9693,E1 24.9107,E2 326.325} C_DIS
LIN {X -62.8835,Y 86.5359,Z 111,A 121.5729,B 24.9281,C -1.9584,E1 24.9055,E2 324.0473} C_DIS
LIN {X -65.4058,Y 84.6448,Z 111,A 123.4435,B 24.9279,C -1.9617,E1 24.9013,E2 322.1621} C_DIS
LIN {X -68.1261,Y 82.4717,Z 111,A 125.2941,B 24.9282,C -1.9571,E1 24.8973,E2 320.3156} C_DIS
LIN {X -71.6422,Y 79.4368,Z 111,A 127.7858,B 24.9286,C -1.9515,E1 24.8921,E2 317.8273} C_DIS
LIN {X -74.1108,Y 77.1379,Z 111,A 129.6875,B 24.9286,C -1.9508,E1 24.8882,E2 315.9194} C_DIS
LIN {X -76.6298,Y 74.638,Z 111,A 131.6665,B 24.9288,C -1.9491,E1 24.8843,E2 313.9362} C_DIS
LIN {X -79.2221,Y 71.8809,Z 111,A 133.7388,B 24.929,C -1.9457,E1 24.8804,E2 311.8629} C_DIS
LIN {X -81.488,Y 69.299,Z 111,A 135.4378,B 24.9298,C -1.9357,E1 24.8773,E2 310.1799} C_DIS
LIN {X -83.8251,Y 66.4531,Z 111,A 137.3158,B 24.9304,C -1.927,E1 24.8741,E2 308.314} C_DIS
LIN {X -87.5527,Y 61.4607,Z 111,A 140.6536,B 24.931,C -1.9178,E1 24.8685,E2 304.9818} C_DIS
LIN {X -89.6212,Y 58.4039,Z 111,A 142.6712,B 24.9313,C -1.9138,E1 24.8654,E2 302.9638} C_DIS
LIN {X -91.8192,Y 54.8832,Z 111,A 145.0665,B 24.9313,C -1.9138,E1 24.8619,E2 300.5562} C_DIS
LIN {X -93.617,Y 51.7563,Z 111,A 146.8978,B 24.932,C -1.9045,E1 24.8594,E2 298.7375} C_DIS
LIN {X -95.2818,Y 48.6212,Z 111,A 148.8621,B 24.9322,C -1.9012,E1 24.8568,E2 296.7706} C_DIS
LIN {X -96.7856,Y 45.5567,Z 111,A 150.8033,B 24.9323,C -1.8998,E1 24.8545,E2 294.8221} C_DIS
LIN {X -98.3193,Y 42.1472,Z 111,A 152.6747,B 24.9331,C -1.8889,E1 24.8524,E2 292.9666} C_DIS
LIN {X -99.5443,Y 39.1609,Z 111,A 154.507,B 24.9332,C -1.8874,E1 24.8505,E2 291.1275} C_DIS
LIN {X -100.7744,Y 35.8803,Z 111,A 156.4602,B 24.9334,C -1.8844,E1 24.8486,E2 289.1705} C_DIS
LIN {X -101.8864,Y 32.5875,Z 111,A 158.4704,B 24.9334,C -1.884,E1 24.8469,E2 287.1496} C_DIS
LIN {X -103.1238,Y 28.433,Z 111,A 160.7049,B 24.9342,C -1.8734,E1 24.8452,E2 284.9274} C_DIS
LIN {X -103.9071,Y 25.4159,Z 111,A 162.314,B 24.9347,C -1.8659,E1 24.8441,E2 283.3268} C_DIS
LIN {X -104.5807,Y 22.4862,Z 111,A 164.0219,B 24.9348,C -1.8643,E1 24.843,E2 281.6127} C_DIS
LIN {X -105.3815,Y 18.3767,Z 111,A 166.0756,B 24.9358,C -1.8502,E1 24.842,E2 279.5807} C_DIS
LIN {X -105.8892,Y 15.1701,Z 111,A 167.9314,B 24.9359,C -1.8489,E1 24.8412,E2 277.7169} C_DIS
LIN {X -106.3413,Y 11.5919,Z 111,A 169.8428,B 24.9364,C -1.8418,E1 24.8406,E2 275.8108} C_DIS
LIN {X -106.7437,Y 6.9641,Z 111,A 172.4153,B 24.9368,C -1.8369,E1 24.84,E2 273.2346} C_DIS
LIN {X -106.941,Y 2.5775,Z 111,A 174.626,B 24.9376,C -1.824,E1 24.8398,E2 271.0413} C_DIS
LIN {X -106.9594,Y -1.5779,Z 111,A 176.955,B 24.9379,C -1.8206,E1 24.8398,E2 268.7063} C_DIS
LIN {X -106.8712,Y -4.6033,Z 111,A 178.7558,B 24.9378,C -1.8221,E1 24.84,E2 266.8913} C_DIS
LIN {X -106.5868,Y -9.0664,Z 111,A -179.0637,B 24.9388,C -1.8064,E1 24.8405,E2 264.735} C_DIS
LIN {X -106.3268,Y -11.7305,Z 111,A -177.4303,B 24.9386,C -1.8092,E1 24.8409,E2 263.0852} C_DIS
LIN {X -105.7767,Y -15.9408,Z 111,A -175.4522,B 24.9399,C -1.7911,E1 24.8417,E2 261.1386} C_DIS
LIN {X -105.2566,Y -19.0711,Z 111,A -173.7329,B 24.9402,C -1.7864,E1 24.8425,E2 259.4201} C_DIS
LIN {X -104.6728,Y -22.0581,Z 111,A -171.9808,B 24.9402,C -1.7858,E1 24.8435,E2 257.6591} C_DIS
LIN {X -104.0345,Y -24.8937,Z 111,A -170.2661,B 24.9402,C -1.7868,E1 24.8446,E2 255.932} C_DIS
LIN {X -103.1749,Y -28.2439,Z 111,A -168.3473,B 24.9404,C -1.7836,E1 24.8459,E2 254.0097} C_DIS
LIN {X -102.0248,Y -32.1532,Z 111,A -166.3522,B 24.9413,C -1.77,E1 24.8475,E2 252.0356} C_DIS
LIN {X -101.2419,Y -34.538,Z 111,A -164.8261,B 24.9411,C -1.7727,E1 24.8489,E2 250.4942} C_DIS
LIN {X -100.0249,Y -37.9164,Z 111,A -162.8444,B 24.9413,C -1.7692,E1 24.8508,E2 248.5096} C_DIS
LIN {X -98.5385,Y -41.6272,Z 111,A -160.8489,B 24.9421,C -1.7576,E1 24.8529,E2 246.5309} C_DIS
LIN {X -97.1903,Y -44.6871,Z 111,A -158.985,B 24.9423,C -1.7551,E1 24.8551,E2 244.6625} C_DIS
LIN {X -95.7391,Y -47.715,Z 111,A -157.2741,B 24.9428,C -1.7468,E1 24.8572,E2 242.9622} C_DIS
LIN {X -94.165,Y -50.7511,Z 111,A -155.3589,B 24.9429,C -1.7449,E1 24.8597,E2 241.0414} C_DIS
LIN {X -92.4714,Y -53.7773,Z 111,A -153.2955,B 24.9428,C -1.7476,E1 24.8626,E2 238.9608} C_DIS
LIN {X -90.6798,Y -56.7435,Z 111,A -151.6621,B 24.9436,C -1.7343,E1 24.8649,E2 237.3506} C_DIS
LIN {X -88.8652,Y -59.5474,Z 111,A -149.7383,B 24.9436,C -1.7348,E1 24.8679,E2 235.4162} C_DIS
LIN {X -86.6697,Y -62.7007,Z 111,A -147.6651,B 24.9439,C -1.7302,E1 24.8713,E2 233.3438} C_DIS
LIN {X -84.5681,Y -65.5054,Z 111,A -145.6455,B 24.9439,C -1.731,E1 24.8747,E2 231.3125} C_DIS
LIN {X -81.7405,Y -69.0027,Z 111,A -142.4717,B 24.9423,C -1.7547,E1 24.8806,E2 228.0677} C_DIS
LIN {X -78.0091,Y -73.1932,Z 111,A -140.648,B 24.9457,C -1.7027,E1 24.8838,E2 226.36} C_DIS
LIN {X -76.124,Y -75.1518,Z 111,A -138.939,B 24.9453,C -1.7092,E1 24.8871,E2 224.6282} C_DIS
LIN {X -73.4316,Y -77.7848,Z 111,A -136.6554,B 24.9449,C -1.7152,E1 24.8918,E2 222.3208} C_DIS
LIN {X -70.671,Y -80.3021,Z 111,A -134.3625,B 24.9444,C -1.7225,E1 24.8967,E2 220.0013} C_DIS
LIN {X -67.64,Y -82.8711,Z 111,A -132.3023,B 24.9448,C -1.7159,E1 24.9011,E2 217.9492} C_DIS
LIN {X -64.7163,Y -85.1751,Z 111,A -130.7054,B 24.946,C -1.6969,E1 24.9046,E2 216.3917} C_DIS
LIN {X -61.8767,Y -87.2583,Z 111,A -128.9512,B 24.9466,C -1.6886,E1 24.9085,E2 214.6511} C_DIS
LIN {X -58.4685,Y -89.5786,Z 111,A -126.7758,B 24.9469,C -1.6837,E1 24.9135,E2 212.4801} C_DIS
LIN {X -55.7269,Y -91.3083,Z 111,A -124.8899,B 24.9467,C -1.6869,E1 24.918,E2 210.5806} C_DIS
LIN {X -52.3346,Y -93.294,Z 111,A -122.7906,B 24.9469,C -1.6837,E1 24.9231,E2 208.4828} C_DIS
LIN {X -49.6945,Y -94.7266,Z 111,A -121.1458,B 24.9469,C -1.683,E1 24.9272,E2 206.8351} C_DIS
LIN {X -46.1717,Y -96.4927,Z 111,A -118.5342,B 24.9458,C -1.7002,E1 24.9339,E2 204.1758} C_DIS
LIN {X -42.5587,Y -98.1399,Z 111,A -116.8581,B 24.9471,C -1.68,E1 24.938,E2 202.5437} C_DIS
LIN {X -38.9041,Y -99.6452,Z 111,A -114.9841,B 24.9478,C -1.6683,E1 24.9428,E2 200.6934} C_DIS
LIN {X -35.9439,Y -100.7521,Z 111,A -113.2831,B 24.9479,C -1.6671,E1 24.9473,E2 198.9919} C_DIS
LIN {X -33.0934,Y -101.7227,Z 111,A -111.4683,B 24.9475,C -1.6738,E1 24.9521,E2 197.1577} C_DIS
LIN {X -29.9658,Y -102.6885,Z 111,A -109.6624,B 24.9475,C -1.6747,E1 24.957,E2 195.3468} C_DIS
LIN {X -26.4105,Y -103.659,Z 111,A -107.8766,B 24.948,C -1.666,E1 24.9618,E2 193.5789} C_DIS
LIN {X -23.5162,Y -104.355,Z 111,A -106.2206,B 24.9479,C -1.6676,E1 24.9663,E2 191.9168} C_DIS
LIN {X -20.2704,Y -105.0322,Z 111,A -104.6547,B 24.9485,C -1.6585,E1 24.9705,E2 190.3708} C_DIS
LIN {X -15.1684,Y -105.8895,Z 111,A -101.986,B 24.9488,C -1.6535,E1 24.9779,E2 187.7115} C_DIS
LIN {X -12.5102,Y -106.2363,Z 111,A -100.1849,B 24.9479,C -1.6679,E1 24.9829,E2 185.8748} C_DIS
LIN {X -9.4779,Y -106.5502,Z 111,A -98.6777,B 24.9482,C -1.6627,E1 24.9871,E2 184.3791} C_DIS
LIN {X -6.218,Y -106.7899,Z 111,A -96.7482,B 24.9477,C -1.67,E1 24.9925,E2 182.4317} C_DIS
LIN {X -2.995,Y -106.9287,Z 111,A -95.0014,B 24.9477,C -1.671,E1 24.9974,E2 180.6823} C_DIS
LIN {X 0.7392,Y -106.965,Z 111,A -93.8184,B 24.9497,C -1.6383,E1 25.0005,E2 179.5768} C_DIS
Enddeposition()
LIN {X 0.7392,Y -106.965,Z 111,A -93.8184,B 24.9497,C -1.6383,E1 25.0005,E2 179.5768} C_DIS
Startdeposition()
$VEL.CP = VEL_PRINT
LIN {X 0.0036,Y -106.0349,Z 111,A -94.4606,B 24.9493,C -1.6448,E1 24.9987,E2 180.2035} C_DIS
LIN {X -3.9134,Y -105.9627,Z 111,A -96.4602,B 24.949,C -1.6492,E1 24.9932,E2 182.193} C_DIS
LIN {X -6.508,Y -105.835,Z 111,A -97.8642,B 24.949,C -1.6491,E1 24.9893,E2 183.5977} C_DIS
LIN {X -9.2904,Y -105.6262,Z 111,A -99.2895,B 24.9488,C -1.6524,E1 24.9853,E2 185.0157} C_DIS
LIN {X -11.6858,Y -105.389,Z 111,A -100.7922,B 24.9493,C -1.6446,E1 24.9811,E2 186.5378} C_DIS
LIN {X -15.6097,Y -104.8794,Z 111,A -102.802,B 24.949,C -1.6501,E1 24.9756,E2 188.5362} C_DIS
LIN {X -18.1418,Y -104.4714,Z 111,A -104.2026,B 24.949,C -1.6499,E1 24.9717,E2 189.9385} C_DIS
LIN {X -20.7036,Y -103.994,Z 111,A -105.6062,B 24.949,C -1.6507,E1 24.9679,E2 191.3419} C_DIS
LIN {X -23.6257,Y -103.3677,Z 111,A -107.0582,B 24.9485,C -1.6578,E1 24.9639,E2 192.7788} C_DIS
LIN {X -25.762,Y -102.8578,Z 111,A -108.4207,B 24.9489,C -1.6516,E1 24.9602,E2 194.158} C_DIS
LIN {X -28.4798,Y -102.1376,Z 111,A -109.8517,B 24.9486,C -1.656,E1 24.9564,E2 195.5807} C_DIS
LIN {X -30.789,Y -101.4664,Z 111,A -111.2356,B 24.9488,C -1.6536,E1 24.9526,E2 196.9725} C_DIS
LIN {X -33.4472,Y -100.6205,Z 111,A -112.5681,B 24.9483,C -1.6616,E1 24.9491,E2 198.2885} C_DIS
LIN {X -35.7212,Y -99.8369,Z 111,A -113.9662,B 24.9484,C -1.6588,E1 24.9454,E2 199.6958} C_DIS
LIN {X -38.3348,Y -98.8618,Z 111,A -115.4824,B 24.9484,C -1.6599,E1 24.9415,E2 201.2127} C_DIS
LIN {X -40.5842,Y -97.9608,Z 111,A -116.8904,B 24.9485,C -1.6574,E1 24.9378,E2 202.6297} C_DIS
LIN {X -43.0073,Y -96.9213,Z 111,A -118.3988,B 24.9486,C -1.6558,E1 24.9339,E2 204.1456} C_DIS
LIN {X -45.9605,Y -95.5543,Z 111,A -120.0541,B 24.9482,C -1.6618,E1 24.9298,E2 205.7908} C_DIS
LIN {X -49.0074,Y -94.0291,Z 111,A -121.8251,B 24.9479,C -1.6668,E1 24.9254,E2 207.5547} C_DIS
LIN {X -51.1272,Y -92.8947,Z 111,A -123.1291,B 24.9479,C -1.6684,E1 24.9222,E2 208.8587} C_DIS
LIN {X -53.3862,Y -91.615,Z 111,A -124.6222,B 24.9479,C -1.6669,E1 24.9186,E2 210.3596} C_DIS
LIN {X -55.7917,Y -90.1692,Z 111,A -126.1983,B 24.9479,C -1.6669,E1 24.9148,E2 211.9406} C_DIS
LIN {X -57.9998,Y -88.7649,Z 111,A -127.454,B 24.9474,C -1.6752,E1 24.9119,E2 213.1809} C_DIS
LIN {X -59.9917,Y -87.4323,Z 111,A -128.9243,B 24.9477,C -1.6706,E1 24.9085,E2 214.6668} C_DIS
LIN {X -62.1207,Y -85.9327,Z 111,A -130.1868,B 24.9472,C -1.6785,E1 24.9056,E2 215.9151} C_DIS
LIN {X -64.3841,Y -84.2488,Z 111,A -131.8661,B 24.9474,C -1.6754,E1 24.9018,E2 217.6078} C_DIS
LIN {X -67.3074,Y -81.9333,Z 111,A -133.7768,B 24.9469,C -1.683,E1 24.8977,E2 219.5075} C_DIS
LIN {X -69.6852,Y -79.9186,Z 111,A -135.4775,B 24.9468,C -1.6857,E1 24.8941,E2 221.2085} C_DIS
LIN {X -72.1748,Y -77.6801,Z 111,A -137.2935,B 24.9465,C -1.689,E1 24.8904,E2 223.0238} C_DIS
LIN {X -74.1244,Y -75.8213,Z 111,A -138.8672,B 24.9466,C -1.6877,E1 24.8872,E2 224.6072} C_DIS
LIN {X -76.4672,Y -73.456,Z 111,A -140.646,B 24.9463,C -1.6923,E1 24.8837,E2 226.3827} C_DIS
LIN {X -79.0194,Y -70.7031,Z 111,A -142.6501,B 24.946,C -1.6978,E1 24.88,E2 228.3826} C_DIS
LIN {X -80.78,Y -68.6848,Z 111,A -144.0937,B 24.9458,C -1.7012,E1 24.8773,E2 229.8245} C_DIS
LIN {X -83.134,Y -65.8159,Z 111,A -146.0538,B 24.9454,C -1.7077,E1 24.8739,E2 231.7785} C_DIS
LIN {X -85.2838,Y -63.0069,Z 111,A -147.9497,B 24.945,C -1.7129,E1 24.8707,E2 233.6709} C_DIS
LIN {X -87.0125,Y -60.5955,Z 111,A -149.4228,B 24.9444,C -1.7217,E1 24.8684,E2 235.1303} C_DIS
LIN {X -88.9856,Y -57.6607,Z 111,A -151.3883,B 24.9443,C -1.7246,E1 24.8653,E2 237.0987} C_DIS
LIN {X -90.2696,Y -55.6309,Z 111,A -152.9204,B 24.9446,C -1.7194,E1 24.863,E2 238.651} C_DIS
LIN {X -91.9573,Y -52.7906,Z 111,A -154.4029,B 24.9436,C -1.7353,E1 24.861,E2 240.1033} C_DIS
LIN {X -93.5177,Y -49.9784,Z 111,A -156.3323,B 24.9437,C -1.733,E1 24.8583,E2 242.0483} C_DIS
LIN {X -94.7995,Y -47.4999,Z 111,A -157.7538,B 24.9432,C -1.7404,E1 24.8566,E2 243.4598} C_DIS
LIN {X -95.8592,Y -45.3256,Z 111,A -159.2465,B 24.9434,C -1.7373,E1 24.8547,E2 244.9681} C_DIS
LIN {X -96.963,Y -42.9128,Z 111,A -160.6634,B 24.9431,C -1.742,E1 24.8531,E2 246.3815} C_DIS
LIN {X -97.9607,Y -40.5845,Z 111,A -161.9857,B 24.9428,C -1.7476,E1 24.8517,E2 247.6977} C_DIS
LIN {X -99.1295,Y -37.6342,Z 111,A -163.57,B 24.9421,C -1.7574,E1 24.8501,E2 249.2675} C_DIS
LIN {X -99.9025,Y -35.5343,Z 111,A -164.8323,B 24.9421,C -1.7591,E1 24.8489,E2 250.533} C_DIS
LIN {X -100.6839,Y -33.2591,Z 111,A -166.3195,B 24.9421,C -1.7562,E1 24.8475,E2 252.0356} C_DIS
LIN {X -101.4685,Y -30.7825,Z 111,A -167.6503,B 24.9417,C -1.7631,E1 24.8464,E2 253.3577} C_DIS
LIN {X -102.3149,Y -27.8333,Z 111,A -169.3412,B 24.9415,C -1.767,E1 24.8452,E2 255.0491} C_DIS
LIN {X -103.1666,Y -24.4962,Z 111,A -171.1916,B 24.9411,C -1.7731,E1 24.8439,E2 256.8957} C_DIS
LIN {X -103.7744,Y -21.7733,Z 111,A -172.6155,B 24.9406,C -1.7808,E1 24.8431,E2 258.3096} C_DIS
LIN {X -104.4746,Y -18.1237,Z 111,A -174.8142,B 24.9406,C -1.7802,E1 24.842,E2 260.5227} C_DIS
LIN {X -104.8902,Y -15.5383,Z 111,A -176.2373,B 24.9403,C -1.7844,E1 24.8414,E2 261.9443} C_DIS
LIN {X -105.3894,Y -11.6828,Z 111,A -178.3688,B 24.9399,C -1.79,E1 24.8406,E2 264.0752} C_DIS
LIN {X -105.6896,Y -8.5264,Z 111,A -179.865,B 24.939,C -1.8033,E1 24.8403,E2 265.5486} C_DIS
LIN {X -105.9163,Y -4.9911,Z 111,A 178.1709,B 24.9388,C -1.8076,E1 24.8399,E2 267.5142} C_DIS
LIN {X -106.0032,Y -2.5921,Z 111,A 176.5951,B 24.9391,C -1.8018,E1 24.8399,E2 269.1133} C_DIS
LIN {X -106.0235,Y 1.4893,Z 111,A 174.506,B 24.9384,C -1.8131,E1 24.8399,E2 271.188} C_DIS
LIN {X -105.9626,Y 3.9135,Z 111,A 173.1465,B 24.9382,C -1.8156,E1 24.8399,E2 272.5499} C_DIS
LIN {X -105.8354,Y 6.5022,Z 111,A 171.7255,B 24.938,C -1.8194,E1 24.8402,E2 273.9703} C_DIS
LIN {X -105.6249,Y 9.3036,Z 111,A 170.2901,B 24.9374,C -1.8273,E1 24.8405,E2 275.3956} C_DIS
LIN {X -105.3884,Y 11.6918,Z 111,A 168.9842,B 24.9371,C -1.8311,E1 24.8409,E2 276.7001} C_DIS
LIN {X -105.0442,Y 14.4542,Z 111,A 167.4717,B 24.9368,C -1.8357,E1 24.8414,E2 278.2107} C_DIS
LIN {X -104.6548,Y 17.0461,Z 111,A 166.1367,B 24.9363,C -1.8432,E1 24.842,E2 279.5357} C_DIS
LIN {X -104.2059,Y 19.6041,Z 111,A 164.724,B 24.936,C -1.8474,E1 24.8427,E2 280.9469} C_DIS
LIN {X -103.6945,Y 22.1506,Z 111,A 163.2151,B 24.936,C -1.8481,E1 24.8435,E2 282.463} C_DIS
LIN {X -103.1208,Y 24.6839,Z 111,A 161.8948,B 24.9355,C -1.8556,E1 24.8444,E2 283.7731} C_DIS
LIN {X -102.4854,Y 27.2021,Z 111,A 160.3887,B 24.9355,C -1.8564,E1 24.8454,E2 285.2862} C_DIS
LIN {X -101.7885,Y 29.7037,Z 111,A 159.0479,B 24.9349,C -1.863,E1 24.8464,E2 286.6189} C_DIS
LIN {X -100.9164,Y 32.5405,Z 111,A 157.4874,B 24.9345,C -1.8697,E1 24.8477,E2 288.1726} C_DIS
LIN {X -100.2612,Y 34.512,Z 111,A 156.2314,B 24.9345,C -1.8684,E1 24.8489,E2 289.4389} C_DIS
LIN {X -99.3866,Y 36.9555,Z 111,A 154.7362,B 24.9345,C -1.8694,E1 24.8503,E2 290.9401} C_DIS
LIN {X -98.3798,Y 39.5552,Z 111,A 153.398,B 24.9337,C -1.8801,E1 24.8516,E2 292.2602} C_DIS
LIN {X -97.382,Y 41.9518,Z 111,A 151.9839,B 24.9335,C -1.884,E1 24.8532,E2 293.6729} C_DIS
LIN {X -96.3259,Y 44.3231,Z 111,A 150.4783,B 24.9335,C -1.8845,E1 24.8549,E2 295.1854} C_DIS
LIN {X -95.2973,Y 46.4954,Z 111,A 149.0931,B 24.9334,C -1.8853,E1 24.8566,E2 296.5763} C_DIS
LIN {X -94.1284,Y 48.8183,Z 111,A 147.5447,B 24.9334,C -1.8843,E1 24.8586,E2 298.1353} C_DIS
LIN {X -92.2515,Y 52.2787,Z 111,A 145.6168,B 24.9325,C -1.8977,E1 24.8612,E2 300.0414} C_DIS
LIN {X -90.846,Y 54.6826,Z 111,A 144.1022,B 24.9322,C -1.9017,E1 24.8633,E2 301.5544} C_DIS
LIN {X -89.5854,Y 56.7263,Z 111,A 142.6478,B 24.9323,C -1.8997,E1 24.8655,E2 303.0208} C_DIS
LIN {X -88.1624,Y 58.9135,Z 111,A 141.3771,B 24.9317,C -1.9087,E1 24.8674,E2 304.2765} C_DIS
LIN {X -86.629,Y 61.1448,Z 111,A 139.9204,B 24.9314,C -1.913,E1 24.8697,E2 305.7301} C_DIS
LIN {X -85.1397,Y 63.2027,Z 111,A 138.374,B 24.9316,C -1.9104,E1 24.8723,E2 307.2902} C_DIS
LIN {X -83.1184,Y 65.8357,Z 111,A 136.6375,B 24.9311,C -1.9173,E1 24.8753,E2 309.0185} C_DIS
LIN {X -81.0692,Y 68.3453,Z 111,A 134.7957,B 24.931,C -1.9186,E1 24.8786,E2 310.8657} C_DIS
LIN {X -78.9381,Y 70.7939,Z 111,A 133.1121,B 24.9305,C -1.9256,E1 24.8817,E2 312.5401} C_DIS
LIN {X -76.7359,Y 73.1772,Z 111,A 131.3074,B 24.9303,C -1.9281,E1 24.8851,E2 314.3467} C_DIS
LIN {X -74.5101,Y 75.4402,Z 111,A 129.7076,B 24.9297,C -1.9365,E1 24.8883,E2 315.9333} C_DIS
LIN {X -72.5699,Y 77.3085,Z 111,A 128.1624,B 24.9297,C -1.9367,E1 24.8914,E2 317.4845} C_DIS
LIN {X -69.4235,Y 80.1471,Z 111,A 125.8812,B 24.9293,C -1.9422,E1 24.8962,E2 319.7615} C_DIS
LIN {X -67.1855,Y 82.0329,Z 111,A 124.1998,B 24.9293,C -1.9421,E1 24.8998,E2 321.4497} C_DIS
LIN {X -64.0497,Y 84.5035,Z 111,A 122.1158,B 24.9288,C -1.9494,E1 24.9044,E2 323.524} C_DIS
LIN {X -61.9383,Y 86.0629,Z 111,A 120.7645,B 24.9284,C -1.9548,E1 24.9074,E2 324.8672} C_DIS
LIN {X -59.7274,Y 87.6113,Z 111,A 119.4499,B 24.9278,C -1.963,E1 24.9104,E2 326.1666} C_DIS
LIN {X -57.6651,Y 88.9828,Z 111,A 118.0458,B 24.9278,C -1.9632,E1 24.9137,E2 327.5749} C_DIS
LIN {X -55.2428,Y 90.5056,Z 111,A 116.5032,B 24.9275,C -1.9662,E1 24.9173,E2 329.1151} C_DIS
LIN {X -52.883,Y 91.9042,Z 111,A 115.0409,B 24.9273,C -1.9696,E1 24.9208,E2 330.5737} C_DIS
LIN {X -49.5365,Y 93.7504,Z 111,A 113.0698,B 24.9267,C -1.9767,E1 24.9256,E2 332.5336} C_DIS
LIN {X -47.485,Y 94.807,Z 111,A 111.6841,B 24.927,C -1.9736,E1 24.9291,E2 333.9306} C_DIS
LIN {X -45.3279,Y 95.8581,Z 111,A 110.1193,B 24.9276,C -1.9656,E1 24.9331,E2 335.5184} C_DIS
LIN {X -42.9714,Y 96.9375,Z 111,A 108.8007,B 24.9272,C -1.9707,E1 24.9364,E2 336.8279} C_DIS
LIN {X -40.5892,Y 97.9587,Z 111,A 107.4718,B 24.9268,C -1.9754,E1 24.9398,E2 338.1487} C_DIS
LIN {X -37.9753,Y 99.0003,Z 111,A 105.9522,B 24.9267,C -1.9775,E1 24.9438,E2 339.6665} C_DIS
LIN {X -35.5385,Y 99.901,Z 111,A 104.4448,B 24.9268,C -1.9754,E1 24.9477,E2 341.182} C_DIS
LIN {X -33.23,Y 100.6933,Z 111,A 103.1423,B 24.9267,C -1.9776,E1 24.9512,E2 342.4816} C_DIS
LIN {X -30.7593,Y 101.4754,Z 111,A 101.7769,B 24.9265,C -1.9805,E1 24.9548,E2 343.8425} C_DIS
LIN {X -28.2688,Y 102.1972,Z 111,A 100.3323,B 24.9265,C -1.9804,E1 24.9587,E2 345.2898} C_DIS
LIN {X -25.7606,Y 102.8582,Z 111,A 99.0016,B 24.9262,C -1.9845,E1 24.9623,E2 346.6127} C_DIS
LIN {X -23.2368,Y 103.4575,Z 111,A 97.5241,B 24.9262,C -1.9829,E1 24.9663,E2 348.096} C_DIS
LIN {X -20.6992,Y 103.9949,Z 111,A 96.1234,B 24.9262,C -1.9841,E1 24.9702,E2 349.4954} C_DIS
LIN {X -18.1372,Y 104.4722,Z 111,A 94.5902,B 24.9265,C -1.9804,E1 24.9744,E2 351.039} C_DIS
LIN {X -14.3075,Y 105.065,Z 111,A 92.5651,B 24.9262,C -1.9844,E1 24.98,E2 353.0561} C_DIS
LIN {X -11.6774,Y 105.3899,Z 111,A 91.2593,B 24.9257,C -1.99,E1 24.9836,E2 354.3494} C_DIS
LIN {X -9.0922,Y 105.6444,Z 111,A 89.77,B 24.9259,C -1.9874,E1 24.9877,E2 355.8457} C_DIS
LIN {X -6.091,Y 105.8581,Z 111,A 88.2291,B 24.9256,C -1.9914,E1 24.992,E2 357.3778} C_DIS
LIN {X -3.7798,Y 105.9669,Z 111,A 87.005,B 24.9256,C -1.9928,E1 24.9954,E2 358.5988} C_DIS
LIN {X -1.1141,Y 106.0281,Z 111,A 85.6254,B 24.9253,C -1.9955,E1 24.9992,E2 359.9719} C_DIS
LIN {X 1.3462,Y 106.0261,Z 111,A 84.1367,B 24.9258,C -1.9896,E1 25.0034,E2 361.4747} C_DIS
LIN {X 3.9082,Y 105.9629,Z 111,A 82.736,B 24.9258,C -1.9891,E1 25.0073,E2 362.8762} C_DIS
LIN {X 6.503,Y 105.8354,Z 111,A 81.3318,B 24.9258,C -1.9891,E1 25.0112,E2 364.2799} C_DIS
LIN {X 9.2863,Y 105.6265,Z 111,A 79.8847,B 24.9256,C -1.9914,E1 25.0153,E2 365.7208} C_DIS
LIN {X 11.7244,Y 105.3845,Z 111,A 78.5881,B 24.9256,C -1.9922,E1 25.0189,E2 367.0145} C_DIS
LIN {X 14.4741,Y 105.0414,Z 111,A 76.9925,B 24.9259,C -1.9881,E1 25.0233,E2 368.6187} C_DIS
LIN {X 17.0524,Y 104.6537,Z 111,A 75.7737,B 24.9254,C -1.9951,E1 25.0266,E2 369.8196} C_DIS
LIN {X 19.6064,Y 104.2055,Z 111,A 74.3743,B 24.9254,C -1.9946,E1 25.0305,E2 371.2186} C_DIS
LIN {X 22.1492,Y 103.6948,Z 111,A 72.7787,B 24.926,C -1.9863,E1 25.0349,E2 372.8319} C_DIS
LIN {X 24.703,Y 103.1162,Z 111,A 71.5595,B 24.9255,C -1.9933,E1 25.0381,E2 374.0329} C_DIS
LIN {X 27.2208,Y 102.4803,Z 111,A 70.0641,B 24.9258,C -1.9888,E1 25.0422,E2 375.5367} C_DIS
LIN {X 29.8479,Y 101.7457,Z 111,A 68.7514,B 24.9254,C -1.9942,E1 25.0457,E2 376.8344} C_DIS
LIN {X 32.2068,Y 101.0244,Z 111,A 67.2614,B 24.926,C -1.9869,E1 25.0497,E2 378.3391} C_DIS
LIN {X 34.4902,Y 100.2688,Z 111,A 65.9511,B 24.926,C -1.9853,E1 25.0532,E2 379.6504} C_DIS
LIN {X 36.9509,Y 99.3883,Z 111,A 64.3661,B 24.9267,C -1.9771,E1 25.0574,E2 381.2516} C_DIS
LIN {X 39.6461,Y 98.3428,Z 111,A 63.1012,B 24.9259,C -1.9875,E1 25.0606,E2 382.4891} C_DIS
LIN {X 42.3418,Y 97.2119,Z 111,A 61.6537,B 24.9257,C -1.9911,E1 25.0643,E2 383.9245} C_DIS
LIN {X 44.3405,Y 96.3177,Z 111,A 60.2404,B 24.9265,C -1.9804,E1 25.0679,E2 385.3596} C_DIS
LIN {X 46.8789,Y 95.1074,Z 111,A 58.8126,B 24.9263,C -1.9823,E1 25.0715,E2 386.7794} C_DIS
LIN {X 49.0009,Y 94.0325,Z 111,A 57.4431,B 24.9267,C -1.9772,E1 25.0749,E2 388.1571} C_DIS
LIN {X 51.1363,Y 92.8896,Z 111,A 56.1381,B 24.9268,C -1.9755,E1 25.0781,E2 389.4623} C_DIS
LIN {X 53.3965,Y 91.609,Z 111,A 54.5703,B 24.9275,C -1.9668,E1 25.0819,E2 391.0459} C_DIS
LIN {X 55.8153,Y 90.1545,Z 111,A 53.3164,B 24.9268,C -1.9756,E1 25.0849,E2 392.2752} C_DIS
LIN {X 57.9878,Y 88.7728,Z 111,A 51.9229,B 24.927,C -1.9733,E1 25.0882,E2 393.6696} C_DIS
LIN {X 59.9919,Y 87.4321,Z 111,A 50.5338,B 24.9274,C -1.9676,E1 25.0914,E2 395.0675} C_DIS
LIN {X 62.1155,Y 85.9365,Z 111,A 49.1345,B 24.9276,C -1.9653,E1 25.0946,E2 396.4672} C_DIS
LIN {X 64.278,Y 84.3305,Z 111,A 47.5297,B 24.9282,C -1.9566,E1 25.0982,E2 398.0868} C_DIS
LIN {X 66.7557,Y 82.3812,Z 111,A 45.963,B 24.928,C -1.9591,E1 25.1016,E2 399.6417} C_DIS
LIN {X 69.2678,Y 80.283,Z 111,A 44.0378,B 24.9288,C -1.9492,E1 25.1057,E2 401.583} C_DIS
LIN {X 71.6914,Y 78.1239,Z 111,A 42.4582,B 24.9285,C -1.9529,E1 25.1089,E2 403.1475} C_DIS
LIN {X 74.0523,Y 75.8925,Z 111,A 40.5415,B 24.9293,C -1.9425,E1 25.1128,E2 405.0807} C_DIS
LIN {X 76.3422,Y 73.5857,Z 111,A 38.9625,B 24.929,C -1.946,E1 25.1159,E2 406.6446} C_DIS
LIN {X 78.5606,Y 71.2154,Z 111,A 37.0495,B 24.9298,C -1.9355,E1 25.1195,E2 408.5742} C_DIS
LIN {X 80.7195,Y 68.7557,Z 111,A 35.4574,B 24.9295,C -1.9387,E1 25.1224,E2 410.1513} C_DIS
LIN {X 82.7898,Y 66.2515,Z 111,A 33.5429,B 24.9303,C -1.9279,E1 25.1258,E2 412.0825} C_DIS
LIN {X 84.5032,Y 64.05,Z 111,A 32.1475,B 24.9303,C -1.9289,E1 25.1282,E2 413.4689} C_DIS
LIN {X 86.0671,Y 61.9324,Z 111,A 30.8235,B 24.9303,C -1.9295,E1 25.1303,E2 414.7852} C_DIS
LIN {X 87.5736,Y 59.7831,Z 111,A 29.348,B 24.9306,C -1.9235,E1 25.1327,E2 416.2676} C_DIS
LIN {X 88.9855,Y 57.661,Z 111,A 28.1324,B 24.9304,C -1.9267,E1 25.1345,E2 417.4697} C_DIS
LIN {X 90.4461,Y 55.3407,Z 111,A 26.6145,B 24.9308,C -1.9212,E1 25.1368,E2 418.9927} C_DIS
LIN {X 91.7134,Y 53.215,Z 111,A 25.2364,B 24.9312,C -1.9159,E1 25.1388,E2 420.3762} C_DIS
LIN {X 92.8968,Y 51.1233,Z 111,A 23.9456,B 24.9314,C -1.9127,E1 25.1405,E2 421.668} C_DIS
LIN {X 94.1203,Y 48.8342,Z 111,A 22.4305,B 24.932,C -1.904,E1 25.1425,E2 423.1954} C_DIS
LIN {X 95.3193,Y 46.4497,Z 111,A 21.1343,B 24.9319,C -1.9062,E1 25.1441,E2 424.4797} C_DIS
LIN {X 96.5404,Y 43.8526,Z 111,A 19.7375,B 24.9317,C -1.9083,E1 25.1457,E2 425.8639} C_DIS
LIN {X 97.5325,Y 41.6005,Z 111,A 18.1271,B 24.9329,C -1.8925,E1 25.1475,E2 427.5027} C_DIS
LIN {X 98.7718,Y 38.5639,Z 111,A 16.3575,B 24.9332,C -1.8875,E1 25.1494,E2 429.2745} C_DIS
LIN {X 99.9015,Y 35.5371,Z 111,A 14.8533,B 24.9329,C -1.8925,E1 25.1508,E2 430.7584} C_DIS
LIN {X 100.6828,Y 33.2624,Z 111,A 13.2857,B 24.9339,C -1.8772,E1 25.1522,E2 432.3532} C_DIS
LIN {X 101.4771,Y 30.7534,Z 111,A 12.0565,B 24.9337,C -1.8811,E1 25.1532,E2 433.5663} C_DIS
LIN {X 102.1984,Y 28.2644,Z 111,A 10.5836,B 24.9342,C -1.8737,E1 25.1543,E2 435.0482} C_DIS
LIN {X 103.1662,Y 24.4977,Z 111,A 8.5766,B 24.9344,C -1.8712,E1 25.1557,E2 437.0494} C_DIS
LIN {X 103.7831,Y 21.7307,Z 111,A 7.1517,B 24.9344,C -1.871,E1 25.1565,E2 438.4665} C_DIS
LIN {X 104.28,Y 19.2057,Z 111,A 5.646,B 24.935,C -1.8617,E1 25.1573,E2 439.9853} C_DIS
LIN {X 104.7159,Y 16.6671,Z 111,A 4.3781,B 24.935,C -1.8626,E1 25.1579,E2 441.2437} C_DIS
LIN {X 105.0992,Y 14.0477,Z 111,A 2.8848,B 24.9355,C -1.8554,E1 25.1585,E2 442.7452} C_DIS
LIN {X 105.4233,Y 11.3586,Z 111,A 1.5736,B 24.9353,C -1.8573,E1 25.1589,E2 444.0443} C_DIS
LIN {X 105.6443,Y 9.0931,Z 111,A 0.1132,B 24.9363,C -1.8434,E1 25.1593,E2 445.5286} C_DIS
LIN {X 105.8354,Y 6.5021,Z 111,A -1.2812,B 24.9366,C -1.8393,E1 25.1596,E2 446.9245} C_DIS
LIN {X 105.9629,Y 3.9073,Z 111,A -2.5939,B 24.9366,C -1.8387,E1 25.1597,E2 448.2309} C_DIS
LIN {X 106.0312,Y 0.7005,Z 111,A -4.3561,B 24.9371,C -1.8318,E1 25.1597,E2 449.9986} C_DIS
LIN {X 106.003,Y -2.6036,Z 111,A -6.0873,B 24.9373,C -1.8283,E1 25.1597,E2 451.7278} C_DIS
LIN {X 105.8891,Y -5.5312,Z 111,A -7.4989,B 24.9372,C -1.8306,E1 25.1595,E2 453.1258} C_DIS
LIN {X 105.7328,Y -7.9862,Z 111,A -8.9792,B 24.9379,C -1.8198,E1 25.1593,E2 454.6227} C_DIS
LIN {X 105.5054,Y -10.5748,Z 111,A -10.5157,B 24.9386,C -1.8095,E1 25.1589,E2 456.1742} C_DIS
LIN {X 105.0364,Y -14.5091,Z 111,A -12.4777,B 24.9386,C -1.8103,E1 25.1582,E2 458.123} C_DIS
LIN {X 104.6517,Y -17.0643,Z 111,A -13.7918,B 24.9386,C -1.8093,E1 25.1576,E2 459.4316} C_DIS
LIN {X 104.2042,Y -19.6128,Z 111,A -15.1793,B 24.9389,C -1.8052,E1 25.1569,E2 460.8206} C_DIS
LIN {X 103.6275,Y -22.4577,Z 111,A -16.7066,B 24.9391,C -1.8019,E1 25.1561,E2 462.3467} C_DIS
LIN {X 103.1226,Y -24.6765,Z 111,A -17.9722,B 24.9395,C -1.7964,E1 25.1553,E2 463.618} C_DIS
LIN {X 102.4807,Y -27.2193,Z 111,A -19.4609,B 24.94,C -1.7888,E1 25.1542,E2 465.116} C_DIS
LIN {X 101.7832,Y -29.7216,Z 111,A -20.7607,B 24.94,C -1.7888,E1 25.1532,E2 466.4084} C_DIS
LIN {X 101.014,Y -32.2387,Z 111,A -22.3281,B 24.9407,C -1.7781,E1 25.1519,E2 467.9922} C_DIS
LIN {X 100.2207,Y -34.6274,Z 111,A -23.6013,B 24.9407,C -1.7775,E1 25.1508,E2 469.2595} C_DIS
LIN {X 99.3652,Y -37.0119,Z 111,A -25.0479,B 24.9413,C -1.7699,E1 25.1494,E2 470.716} C_DIS
LIN {X 98.3711,Y -39.5766,Z 111,A -26.3551,B 24.9411,C -1.773,E1 25.1481,E2 472.0087} C_DIS
LIN {X 97.3839,Y -41.9473,Z 111,A -27.8022,B 24.9415,C -1.7662,E1 25.1465,E2 473.4638} C_DIS
LIN {X 96.3178,Y -44.3404,Z 111,A -29.2386,B 24.9419,C -1.761,E1 25.1448,E2 474.9047} C_DIS
LIN {X 95.2898,Y -46.5108,Z 111,A -30.61,B 24.9423,C -1.7539,E1 25.1431,E2 476.2855} C_DIS
LIN {X 94.0178,Y -49.0288,Z 111,A -32.0346,B 24.9423,C -1.7536,E1 25.1413,E2 477.7032} C_DIS
LIN {X 92.8927,Y -51.1307,Z 111,A -33.3231,B 24.9426,C -1.7498,E1 25.1396,E2 478.994} C_DIS
LIN {X 91.6124,Y -53.3909,Z 111,A -34.7998,B 24.9431,C -1.7426,E1 25.1376,E2 480.4801} C_DIS
LIN {X 90.1753,Y -55.782,Z 111,A -36.1393,B 24.9429,C -1.7454,E1 25.1356,E2 481.8061} C_DIS
LIN {X 88.7657,Y -57.9986,Z 111,A -37.5326,B 24.9431,C -1.7425,E1 25.1335,E2 483.1993} C_DIS
LIN {X 87.4308,Y -59.9938,Z 111,A -38.915,B 24.9436,C -1.7352,E1 25.1313,E2 484.5921} C_DIS
LIN {X 85.9377,Y -62.1138,Z 111,A -40.3102,B 24.9438,C -1.7315,E1 25.1291,E2 485.9891} C_DIS
LIN {X 84.2792,Y -64.3446,Z 111,A -41.9613,B 24.9445,C -1.7211,E1 25.1263,E2 487.6569} C_DIS
LIN {X 82.003,Y -67.2224,Z 111,A -43.8299,B 24.9445,C -1.7207,E1 25.123,E2 489.5178} C_DIS
LIN {X 80.2183,Y -69.3419,Z 111,A -45.4284,B 24.945,C -1.7125,E1 25.1201,E2 491.1284} C_DIS
LIN {X 77.9417,Y -71.8899,Z 111,A -47.2181,B 24.9452,C -1.7102,E1 25.1167,E2 492.9156} C_DIS
LIN {X 75.7785,Y -74.1677,Z 111,A -48.949,B 24.9456,C -1.7045,E1 25.1134,E2 494.6525} C_DIS
LIN {X 73.1651,Y -76.7477,Z 111,A -50.933,B 24.9459,C -1.6997,E1 25.1094,E2 496.6395} C_DIS
LIN {X 70.653,Y -79.0643,Z 111,A -52.7007,B 24.9459,C -1.6987,E1 25.1057,E2 498.4025} C_DIS
LIN {X 67.8207,Y -81.5068,Z 111,A -54.6333,B 24.9459,C -1.6978,E1 25.1016,E2 500.3296} C_DIS
LIN {X 65.6579,Y -83.2589,Z 111,A -56.1903,B 24.9463,C -1.6923,E1 25.0982,E2 501.8938} C_DIS
LIN {X 63.0046,Y -85.2855,Z 111,A -57.9011,B 24.9463,C -1.6923,E1 25.0944,E2 503.5984} C_DIS
LIN {X 60.9012,Y -86.8001,Z 111,A -59.2955,B 24.9465,C -1.6897,E1 25.0912,E2 504.9942} C_DIS
LIN {X 58.9215,Y -88.1569,Z 111,A -60.6763,B 24.9469,C -1.6836,E1 25.088,E2 506.3848} C_DIS
LIN {X 56.7197,Y -89.5895,Z 111,A -62.0012,B 24.9469,C -1.6848,E1 25.0849,E2 507.7025} C_DIS
LIN {X 54.3431,Y -91.0495,Z 111,A -63.5024,B 24.9469,C -1.6822,E1 25.0813,E2 509.2052} C_DIS
LIN {X 52.0968,Y -92.3532,Z 111,A -64.8181,B 24.9469,C -1.6833,E1 25.0782,E2 510.5143} C_DIS
LIN {X 49.9725,Y -93.5208,Z 111,A -66.3054,B 24.9475,C -1.6736,E1 25.0745,E2 512.0202} C_DIS
LIN {X 47.6719,Y -94.7143,Z 111,A -67.7788,B 24.9478,C -1.6683,E1 25.0708,E2 513.5023} C_DIS
LIN {X 45.1038,Y -95.9625,Z 111,A -69.1671,B 24.9476,C -1.6722,E1 25.0673,E2 514.8776} C_DIS
LIN {X 42.8988,Y -96.9691,Z 111,A -70.6043,B 24.9481,C -1.6649,E1 25.0636,E2 516.3285} C_DIS
LIN {X 39.3571,Y -98.4602,Z 111,A -72.5952,B 24.9481,C -1.6654,E1 25.0585,E2 518.3136} C_DIS
LIN {X 36.7537,Y -99.4603,Z 111,A -74.0164,B 24.9479,C -1.6669,E1 25.0548,E2 519.7283} C_DIS
LIN {X 34.4889,Y -100.2692,Z 111,A -75.3119,B 24.948,C -1.6654,E1 25.0514,E2 521.0248} C_DIS
LIN {X 31.8322,Y -101.143,Z 111,A -76.7698,B 24.948,C -1.6657,E1 25.0475,E2 522.4791} C_DIS
LIN {X 29.4667,Y -101.858,Z 111,A -78.1452,B 24.9482,C -1.6626,E1 25.0438,E2 523.8596} C_DIS
LIN {X 26.8006,Y -102.5909,Z 111,A -79.5462,B 24.9481,C -1.6648,E1 25.0401,E2 525.2532} C_DIS
LIN {X 23.2235,Y -103.4605,Z 111,A -81.7065,B 24.9486,C -1.6559,E1 25.0341,E2 527.4315} C_DIS
LIN {X 20.6958,Y -103.9956,Z 111,A -83.0966,B 24.9486,C -1.6549,E1 25.0303,E2 528.8222} C_DIS
LIN {X 18.157,Y -104.4686,Z 111,A -84.5004,B 24.9488,C -1.6534,E1 25.0265,E2 530.2279} C_DIS
LIN {X 15.5541,Y -104.8879,Z 111,A -85.9189,B 24.9488,C -1.6526,E1 25.0226,E2 531.6469} C_DIS
LIN {X 12.7888,Y -105.2599,Z 111,A -87.4772,B 24.949,C -1.6497,E1 25.0182,E2 533.211} C_DIS
LIN {X 9.0875,Y -105.6448,Z 111,A -89.4326,B 24.949,C -1.6508,E1 25.0128,E2 535.1626} C_DIS
LIN {X 6.4968,Y -105.8357,Z 111,A -90.8351,B 24.949,C -1.6502,E1 25.0089,E2 536.5659} C_DIS
LIN {X 3.8998,Y -105.9632,Z 111,A -92.1566,B 24.9488,C -1.653,E1 25.0052,E2 537.8803} C_DIS
LIN {X 0.7334,Y -106.0305,Z 111,A -93.5877,B 24.9481,C -1.6638,E1 25.0013,E2 539.2857} C_DIS
Enddeposition()
LIN {X 0.7859,Y -112.3805,Z 112,A -93.0438,B 24.9531,C -1.5826,E1 25.0023,E2 538.9343} C_DIS
Startdeposition()
$VEL.CP = VEL_PRINT
LIN {X 3.4288,Y -112.3316,Z 112,A -91.6439,B 24.9529,C -1.5853,E1 25.0062,E2 537.5283} C_DIS
LIN {X 6.1845,Y -112.2136,Z 112,A -90.2388,B 24.9529,C -1.5858,E1 25.0101,E2 536.1224} C_DIS
LIN {X 8.9365,Y -112.028,Z 112,A -88.834,B 24.9529,C -1.5864,E1 25.014,E2 534.7169} C_DIS
LIN {X 11.6831,Y -111.775,Z 112,A -87.4381,B 24.9529,C -1.5867,E1 25.0179,E2 533.3211} C_DIS
LIN {X 14.4596,Y -111.4498,Z 112,A -85.9986,B 24.9527,C -1.5882,E1 25.0219,E2 531.8791} C_DIS
LIN {X 17.1536,Y -111.0671,Z 112,A -84.6209,B 24.9527,C -1.5888,E1 25.0257,E2 530.5014} C_DIS
LIN {X 19.8741,Y -110.6127,Z 112,A -83.2173,B 24.9527,C -1.5898,E1 25.0296,E2 529.0969} C_DIS
LIN {X 22.6191,Y -110.0841,Z 112,A -81.8118,B 24.9527,C -1.5902,E1 25.0334,E2 527.6922} C_DIS
LIN {X 25.3139,Y -109.4959,Z 112,A -80.4083,B 24.9526,C -1.5914,E1 25.0373,E2 526.2878} C_DIS
LIN {X 27.9575,Y -108.8509,Z 112,A -79.0068,B 24.9524,C -1.5934,E1 25.0411,E2 524.8836} C_DIS
LIN {X 30.6204,Y -108.132,Z 112,A -77.6126,B 24.9524,C -1.5944,E1 25.0448,E2 523.4893} C_DIS
LIN {X 33.2648,Y -107.348,Z 112,A -76.2011,B 24.9523,C -1.5963,E1 25.0486,E2 522.0758} C_DIS
Enddeposition()
END
